(* CODESYS project Motor_4.2.6.0.library
   Company: ESO
   Description: Local Device Control - LDC Motor Library based on State Machine
   Version: 4.2.6.0
   Placeholder: ESO LDC Motor Library
   Author: Dan Popovic
   Title: ESO LDC Motor Library

Project tree, tasks and I/O mapping:
  libraries: ESO LDC Common Library, * (ESO); ESO LDC Timer Library, * (ESO); ESO MUDPI Library, * (ESO); Tc2_EtherCAT, * (Beckhoff Automation GmbH); Tc2_IoFunctions, * (Beckhoff Automation GmbH); Tc2_Math, * (Beckhoff Automation GmbH); Tc2_MC2, * (Beckhoff Automation GmbH); Tc2_MC2_Drive, * (Beckhoff Automation GmbH); Tc2_NC, * (Beckhoff Automation GmbH); Tc2_Standard, * (Beckhoff Automation GmbH); Tc2_System, * (Beckhoff Automation GmbH); Tc2_Utilities, * (Beckhoff Automation GmbH); Tc3_EventLogger, * (Beckhoff Automation GmbH); Tc3_Module, * (Beckhoff Automation GmbH); VisuDialogs, * (System); VisuSymbols, 3.5.10.0 (System)
  config/
    Mapping_with_new_EL6688_09_05.xml
    Mapping_with_old_EL6688_03_03.xml
    Mappings_SIM.xml
  00000000-0000-0000-0000-000000000000|config\Mapping_with_new_EL6688_09_05.xml
  00000000-0000-0000-0000-000000000000|config\Mapping_with_old_EL6688_03_03.xml
  00000000-0000-0000-0000-000000000000|config\Mappings_SIM.xml
  doc/
    AM8121_0F20_0000.xti
    EL7041_Phytron_57_500_1.2.xti
    EL7201_9014___AM8121_0F20_0000.xti
    MotorStateMachine.jpg
    Phytron_57_500_1.2_PID.xti
  00000000-0000-0000-0000-000000000000|doc\AM8121_0F20_0000.xti
  00000000-0000-0000-0000-000000000000|doc\EL7041_Phytron_57_500_1.2.xti
  00000000-0000-0000-0000-000000000000|doc\EL7201_9014___AM8121_0F20_0000.xti
  00000000-0000-0000-0000-000000000000|doc\MotorStateMachine.jpg
  00000000-0000-0000-0000-000000000000|doc\Phytron_57_500_1.2_PID.xti
  DUTs/
    Enumerated/
      Common/
        data type E_TIME_MODE
      Motor/
        data type E_DIRECTION
        data type E_MOTOR_AXIS_TYPE
        data type E_MOTOR_COMMAND
        data type E_MOTOR_ERROR
        data type E_MOTOR_EVENT
        data type E_MOTOR_INIT_ACTION
        data type E_MOTOR_INIT_SEQ_STATE
        data type E_MOTOR_INIT_STATE
        data type E_MOTOR_MODE
        data type E_MOTOR_MOVE_TYPE
        data type E_MOTOR_MOVING_STATE
        data type E_MOTOR_POST_INIT_STATE
        data type E_MOTOR_PRE_INIT_STATE
        data type E_MOTOR_RESET_STATE
        data type E_MOTOR_RPC_ERROR
        data type E_MOTOR_STATE
        data type E_MOTOR_STATUS
        data type E_MOTOR_SUBSTATE
        data type E_MOTOR_SWITCH_INDEX
      MultiAxis/
        data type E_MA_ADC_MOUNTING
        data type E_MA_AXES_ID
        data type E_MA_COMMAND
        data type E_MA_EVENT
        data type E_MA_MODE
        data type E_MA_ROTATOR_TYPE
        data type E_MA_RPC_ERROR
        data type E_MA_STATE
        data type E_MA_SUBSTATE
      Tracking/
        data type E_ADC_AXES_ID
        data type E_ADC_MODE
        data type E_DROT_MODE
        data type E_TRK_COMMAND
    Interfaces/
      interface ITrackCtrl: ComputeNextPos, HandleStates, Init, IsError, MoveInPos, MoveInSpeed, Reset
    Structures/
      Astro/
        data type E_ASTRO_TELESCOPE
        data type T_ASTRO_CCS_DATA
        data type T_ASTRO_DATA
        data type T_ASTRO_EL6688_DATA
        data type T_ASTRO_ENVIRONMENT
        data type T_ASTRO_MEAN_COORDINATES
        data type T_ASTRO_POLAR_MOTION
        data type T_ASTRO_SITE_CONSTANTS
        data type T_ASTRO_TIME
        data type T_ASTRO_TRACKING_DATA
      CCS_Sim/
        data type T_CCS_CFG
        data type T_CCS_CTRL
        data type T_CCS_STAT
      Common/
        data type T_PTP_TIME
        data type T_TIMEVAL
        data type T_UTC_TIME
      Motor/
        data type T_MOTOR_ACTIVE_LOW
        data type T_MOTOR_AXIS_CFG
        data type T_MOTOR_CFG
        data type T_MOTOR_CTRL
        data type T_MOTOR_INFO
        data type T_MOTOR_INIT_STEP
        data type T_MOTOR_MC_PARAMETER
        data type T_MOTOR_MOTION
        data type T_MOTOR_SIGNAL
        data type T_MOTOR_SPEED
        data type T_MOTOR_STAT
        data type T_MOTOR_SWITCHES
        data type T_POSITION
      MultiAxis/
        data type T_MA_CFG
        data type T_MA_CTRL
        data type T_MA_SM_STAT
        data type T_MA_STAT
        data type T_MA_TOUT_CFG
      Simulation/
        data type T_SIM_MOTOR_CFG
        data type T_SIM_MOTOR_STAT
      Tracking/
        data type T_ADC_CFG
        data type T_ADC_CMD
        data type T_ADC_CTRL
        data type T_ADC_INFO
        data type T_ADC_STAT
        data type T_ADC_UNIT_CFG
        data type T_ASTRO_COORDINATES
        data type T_DROT_CFG
        data type T_DROT_CTRL
        data type T_DROT_INFO
        data type T_DROT_STAT
  GVLs/
    global variables GVL_TrkDefaultEnvironment
    global variables GVL_TrkSiteConstants
  lib/
  POUs/
    Astro/
      function block FB_ASTRO [ST]: M_AstroDataUpdate, M_Configure, M_GetDec_ddmmss, M_GetRa_hhmmss, M_OffsetRaDec_arcsec, M_SetRaDec_hdmmss, M_TrkUpdate
    Functions/
      function F_astroDms2rad [ST]
      function F_astroHms2rad [ST]
      function F_astroRad2Dms [ST]
      function F_astroRad2Hms [ST]
      function F_astroSplitHms [ST]
      function F_atan2 [ST]
      function F_DCTIME64_TO_ULINT [ST]
      function F_MOD [ST]
      function F_RAD2DMS_STRING [ST]
      function F_RAD2HMS_STRING [ST]
      function F_slaPa [ST]
      function F_timeGetAbsoluteDcTime [ST]
      function F_timeGetDcTime [ST]
      function F_timeGetUTC [ST]
      function F_timeUTCToJD [ST]
      function F_timeUTCToMJD [ST]
      function F_vltMod [ST]
      function F_vltSign [ST]
    Misc/
      function block FB_DIGITAL_SIGNAL_FILTER [ST]
    Motor/
      function block FB_MOTOR [ST]: ActionClearNOVRAM, ActionErrExecute, ActionInitAbort, ActionInitComplete, ActionInitExecute, ActionInitReject, ActionMoveExecute, ActionResetExecute, ActionSetPosition, ActionStopExecute, ActionUnexpExecute, ActivityClearingNOVRAM, ActivityInitAborting, ActivityInitializing, ActivityMoving, ActivitySettingPosition, ActivityStopping, CheckForEvents, Dummy_UserExample, M_Configure, M_GetActualPos, M_GetOptimisedDistance, M_GetOptimisedPosition, M_GetRpcErrorText, M_HandleEnabled, M_MotorBrakeControl, M_MotorInitLock, M_MotorInitSeq, M_MotorPostInit, M_MotorPreInit, M_MotorReset, M_NormalizePos, M_NOVRAM_Clear, M_NOVRAM_Load, M_NOVRAM_Save, M_SetError, M_SetRpcStatus, M_UpdateSwitches, RPC_Disable, RPC_Enable, RPC_Init, RPC_MoveAbs, RPC_MoveRel, RPC_MoveVel, RPC_Reset, RPC_SetDebug, RPC_SetLog, RPC_Stop, UserPostInit, UserPostMove, UserPreInit, UserPreMove
      function block FB_MOTOR_BASE [ST]: ActionClearNOVRAM, ActionEnableExecute, ActionErrExecute, ActionInitAbort, ActionInitComplete, ActionInitExecute, ActionInitReject, ActionMoveExecute, ActionResetExecute, ActionSetPosition, ActionStopExecute, ActionUnexpExecute, ActivityClearingNOVRAM, ActivityInitAborting, ActivityInitializing, ActivityMoving, ActivitySettingPosition, ActivityStopping, CheckForEvents, M_CheckDisableIfUnsafe, M_GetErrorText, M_GetLogicalState, M_GetTimeInSec, M_LogEventDebug, M_LogEventEnd, M_LogEventError, M_LogEventGeneral, M_LogEventMoveAbs, M_LogEventMoveRel, M_LogEventMoveVel, M_LogEventStart, M_ReportFirstError, M_SetStatus, M_SetStatusDescription, ProcessEvents, SetAction, SetEvent, SetState, SetStatus
      function block FB_SIM_MOTOR [ST]: GetLogicalState, RPC_ResetConfig, RPC_SetCouplerState, RPC_SetDelay_Brake, RPC_SetDelay_SwitchActive, RPC_SetDelay_SwitchFind, RPC_SetFailure_BrakeFeedback
    MultiAxis/
      function block FB_MA_ADC [ST]: M_LogCommand, RPC_Disable, RPC_Enable, RPC_Init, RPC_MoveAbs, RPC_MoveAngle, RPC_MoveRel, RPC_MoveVel, RPC_Reset, RPC_StartTrack, RPC_Stop, RPC_StopTrack, User_ComputeAutoPos, User_ComputeNextPos, User_Configure, User_GetParams, User_SetParams
      function block FB_MA_BASE [ST]: ActionDisableExecute, ActionEnableExecute, ActionInitExecute, ActionMoveAbsExecute, ActionMoveVelExecute, ActionResetExecute, ActionStopExecute, ActionTrackExecute, ActivityDisabling, ActivityEnabling, ActivityInitialising, ActivityMoving, ActivityPresetting, ActivityResetting, ActivityStopping, ActivityTracking, CheckForEvents, M_AxesIdle, M_AxesInitialised, M_CheckAxesState, M_CheckError, M_Configure, M_GetMaxPosError, M_GetRpcErrorText, M_HomeMotors, M_LogCommand, M_LogEventError, M_LogEventGeneral, M_NextMove, M_NextMoveAbs, M_RestartTimer, M_SetInit, M_SetMode, M_SetRpcStatus, M_SetStatus, ProcessEvents, RPC_Init, SetAction, SetEvent, SetState, User_ComputeNextPos, User_Configure, User_GetParams, User_SetParams
      function block FB_MA_DROT [ST]: M_LogCommand, RPC_Disable, RPC_Enable, RPC_Init, RPC_MoveAbs, RPC_MoveAngle, RPC_MoveRel, RPC_MoveVel, RPC_Reset, RPC_StartTrack, RPC_Stop, RPC_StopTrack, RPC_TrackOffset, User_ComputeNextPos, User_Configure, User_GetParams, User_SetParams
      function block FB_TRK_BASE [ST]: User_Configure, User_GetParams, User_SetParams
    program MAIN [ST]
  Version/
    global variables Global_Version
  VISUs/
    Astro/
      visualisation GUI_ASTRO_CCS_SIM
    Motor/
      visualisation GUI_Motor001_Cfg
      visualisation GUI_Motor001_Ctrl
      visualisation GUI_Motor002_Cfg
      visualisation GUI_Motor002_Ctrl
    Templates/
      visualisation GUI_TEMPLATE_ASTRO_CCS_SIM
      visualisation GUI_TEMPLATE_MA_ADC
      visualisation GUI_TEMPLATE_MA_DROT
      visualisation GUI_TEMPLATE_MOTOR_CONFIG
      visualisation GUI_TEMPLATE_MOTOR_CONTROL
    Tracking/
      visualisation GUI_ADC_Motor1
      visualisation GUI_ADC_Motor2
      visualisation GUI_DROT_Cfg
      visualisation GUI_DROT_Motor
      visualisation GUI_MA_ADC
      visualisation GUI_MA_DROT
      visualisation GUI_TIMER
  global variables GCL
  text list GlobalTextList
  global variables GPL
*)

// DUTs/Enumerated/Common/E_TIME_MODE
{attribute 'qualified_only'}
{attribute 'strict'}
TYPE E_TIME_MODE :
(
	LOCAL	:= 0,
	UTC		:= 1
);
END_TYPE

// DUTs/Enumerated/Motor/E_DIRECTION
{attribute 'qualified_only'}
{attribute 'strict'}
TYPE E_DIRECTION :
(
	NEGATIVE := 1,
	POSITIVE
);
END_TYPE

// DUTs/Enumerated/Motor/E_MOTOR_AXIS_TYPE
{attribute 'qualified_only'}
{attribute 'strict'}
TYPE E_MOTOR_AXIS_TYPE :
(
	LINEAR				:= 1,
	CIRCULAR,
	CIRCULAR_OPTIMISED
);
END_TYPE

// DUTs/Enumerated/Motor/E_MOTOR_COMMAND
{attribute 'qualified_only'}
{attribute 'strict'}
TYPE E_MOTOR_COMMAND :
(
	NONE	:= 0,
	
	// Commands corresponding to events - MUST match E_MOTOR_EVENT !!!
	RESET,
	INIT,
	STOP,
	ENABLE,
	DISABLE,
	MOTOR_MOVE,
	SET_POSITION,
	CLEAR_NOVRAM
);
END_TYPE

// DUTs/Enumerated/Motor/E_MOTOR_ERROR
{attribute 'qualified_only'}
// 'strict' cannot be used since we mix our own codes with TC codes
//{attribute 'strict'}
TYPE E_MOTOR_ERROR :
(
	OK					:= 0,
	HW_NOT_OP,			
	LOCAL,			
	INIT_ABORTED,		
	TIMEOUT_INIT,
	TIMEOUT_MOVE,
	TIMEOUT_RESET,
	TIMEOUT_SETPOS,
	TIMEOUT_USER_PREINIT,
	TIMEOUT_USER_POSTINIT,
	TIMEOUT_USER_PREMOVE,
	TIMEOUT_USER_POSTMOVE,
	SETPOS,
	STOP,
	
	ABORT,
	SW_LIMIT_LOWER,
	SW_LIMIT_UPPER,
	BRAKE_ACTIVE,
	BRAKE_ENGAGE,
	BRAKE_DISENGAGE,
	SWITCH_NOT_USED,
	ENABLE,
	NOVRAM_READ,
	NOVRAM_WRITE,
	SWITCH_EXIT,
	STOP_LIMITS_BOTH,
	HW_LIMITS_BOTH,
	IN_POS,
	LOCKED,
	SoE_ADS_ERROR,
	SoE_SERCOS_ERROR,
	
	UNSAFE,		// EICSSW-1923

	// Simulator errors
	SIM_NOT_INITIALISED			:= 90,
	SIM_NULL_POINTER			:= 100,	

	// TwinCAT errors
	TC_VEL						:= 16929,	
	TC_NOT_READY_FOR_START		:= 16933,	
	TC_DISABLED_MOVE			:= 16992,	
	TC_BISECTION				:= 17022,	
	TC_MODULO_POS				:= 17026,	
	TC_STOP_ACTIVE				:= 17135,	
	TC_VEL_NEG					:= 17241,	
	TC_TARGET_LSW				:= 17504,	
	TC_TARGET_USW				:= 17505,	
	TC_FOLLOWING_ERROR			:= 17744,	
	TC_NOT_READY				:= 18000,	
	TC_IN_POS_6_SEC				:= 19207	

);
END_TYPE

// DUTs/Enumerated/Motor/E_MOTOR_EVENT
{attribute 'qualified_only'}
{attribute 'strict'}
TYPE E_MOTOR_EVENT :
(
	NONE	:= 0,
	
	(* events corresponding to commands - MUST match E_MOTOR_COMMAND *)
	RESET,
	INIT,
	STOP,
	ENABLE,
	DISABLE,
	MOTOR_MOVE,
	SET_POSITION,
	CLEAR_NOVRAM,
	
	(* 
		Events corresponding to internal events 
	*)
	
	MOVEDONE,		// Needed for detection of HW failures during initialisation
	STOPDONE,
	ENABLEDONE,
	DISABLEDONE,
	INITDONE,
	SETPOSDONE,
	

	HWOK,
	ERRLOCAL,
	ERRHW,
	ERRRESET,
	ERRFAULT,
	ERRINIT,
	ERRSTOP,
	ERRENABLE,
	ERRDISABLE,
	ERRBRAKE,
	ERRINPOS,
	ERRLOCKED,
	ERRTARGETPAR,
	ERRUSERPREINIT,
	ERRUSERPREMOVE,
	ERRUSERPOSTINIT,
	ERRUSERPOSTMOVE,
	TIMEOUT_MOVE,
	TIMEOUT_SETPOS,
	SW_LIMIT_LOWER,
	SW_LIMIT_UPPER,
	
	UNSAFE		// EICSSW-1923
	
);
END_TYPE

// DUTs/Enumerated/Motor/E_MOTOR_INIT_ACTION
TYPE E_MOTOR_INIT_ACTION :
(
	MOTOR_INIT_ACTION_END				:= 0,
	MOTOR_INIT_ACTION_FIND_INDEX,
	MOTOR_INIT_ACTION_FIND_REF_LE,
	MOTOR_INIT_ACTION_FIND_REF_UE,
	MOTOR_INIT_ACTION_FIND_LHW,
	MOTOR_INIT_ACTION_FIND_UHW,
	MOTOR_INIT_ACTION_DELAY,
	MOTOR_INIT_ACTION_MOVE_ABS,
	MOTOR_INIT_ACTION_MOVE_REL,
	MOTOR_INIT_ACTION_CALIB_ABS,
	MOTOR_INIT_ACTION_CALIB_REL,
	MOTOR_INIT_ACTION_CALIB_SWITCH,
	// The following steps cannot be configured in the INIT sequence
	MOTOR_INIT_ACTION_STEP1_START,
	MOTOR_INIT_ACTION_STEP1_EXECUTE,
	MOTOR_INIT_ACTION_STEP2_START,
	MOTOR_INIT_ACTION_STEP2_EXECUTE,
	MOTOR_INIT_ACTION_STOP
);
END_TYPE

// DUTs/Enumerated/Motor/E_MOTOR_INIT_SEQ_STATE
TYPE E_MOTOR_INIT_SEQ_STATE :
(
	MOTOR_INIT_SEQ_STATE_START				:= 0,
	MOTOR_INIT_SEQ_STATE_EXECUTE,
	MOTOR_INIT_SEQ_STATE_END
);
END_TYPE

// DUTs/Enumerated/Motor/E_MOTOR_INIT_STATE
TYPE E_MOTOR_INIT_STATE :
(
	MOTOR_INIT_STATE_START				:= 0,
	MOTOR_INIT_STATE_RESET,
	MOTOR_INIT_STATE_WAIT_READY,
	MOTOR_INIT_STATE_PRE_INIT,
	MOTOR_INIT_STATE_USER_PRE_INIT,
	MOTOR_INIT_STATE_INIT_SEQ,
	MOTOR_INIT_STATE_INIT_LOCK,
	MOTOR_INIT_STATE_POST_INIT,
	MOTOR_INIT_STATE_USER_POST_INIT,
	MOTOR_INIT_STATE_WAIT_BRAKE,
	MOTOR_INIT_STATE_SAVE_NOVRAM,
	MOTOR_INIT_STATE_END
);
END_TYPE

// DUTs/Enumerated/Motor/E_MOTOR_MODE
{attribute 'qualified_only'}
{attribute 'strict'}
TYPE E_MOTOR_MODE :
(
	POS				:= 0,
	VEL
);
END_TYPE

// DUTs/Enumerated/Motor/E_MOTOR_MOVE_TYPE
{attribute 'qualified_only'}
{attribute 'strict'}
TYPE E_MOTOR_MOVE_TYPE :
(
	NONE	:= 0,
	
	ABSOLUTE,
	RELATIVE,
	VELOCITY,
	TRACKING

);
END_TYPE

// DUTs/Enumerated/Motor/E_MOTOR_MOVING_STATE
TYPE E_MOTOR_MOVING_STATE :
(
	MOTOR_MOVING_STATE_NONE	:= 0,
	MOTOR_MOVING_STATE_ENABLE,
	MOTOR_MOVING_STATE_WAIT_BRAKES,
	MOTOR_MOVING_STATE_USER_PRE_MOVE,
	MOTOR_MOVING_STATE_WAIT_ABSOLUTE,
	MOTOR_MOVING_STATE_WAIT_OPTIMISED,
	MOTOR_MOVING_STATE_WAIT_VELOCITY,
	MOTOR_MOVING_STATE_USER_POST_MOVE,
	MOTOR_MOVING_STATE_APPLY_BRAKES,
	MOTOR_MOVING_STATE_DISABLE,
	MOTOR_MOVING_STATE_CHECK_IN_POS,
	MOTOR_MOVING_STATE_END
);
END_TYPE

// DUTs/Enumerated/Motor/E_MOTOR_POST_INIT_STATE
TYPE E_MOTOR_POST_INIT_STATE :
(
	MOTOR_POST_INIT_STATE_START	:= 0,
	MOTOR_POST_INIT_STATE_WRITE,
	MOTOR_POST_INIT_STATE_END
);
END_TYPE

// DUTs/Enumerated/Motor/E_MOTOR_PRE_INIT_STATE
TYPE E_MOTOR_PRE_INIT_STATE :
(
	MOTOR_PRE_INIT_STATE_START	:= 0,
	MOTOR_PRE_INIT_STATE_READ,
	MOTOR_PRE_INIT_STATE_GET_USER_UNITS,
	MOTOR_PRE_INIT_STATE_WRITE,
	MOTOR_PRE_INIT_STATE_END
);
END_TYPE

// DUTs/Enumerated/Motor/E_MOTOR_RESET_STATE
TYPE E_MOTOR_RESET_STATE :
(
	MOTOR_RESET_STATE_START	:= 0,
	MOTOR_RESET_STATE_SoE_RESET,
	MOTOR_RESET_STATE_SoE_WAIT_RESET,
	MOTOR_RESET_STATE_RESET_AXIS,
	MOTOR_RESET_STATE_WAIT,
	MOTOR_RESET_STATE_END
);
END_TYPE

// DUTs/Enumerated/Motor/E_MOTOR_RPC_ERROR
{attribute 'qualified_only'}
{attribute 'strict'}
TYPE E_MOTOR_RPC_ERROR :
(
	OK						:= 0,
	NOT_OP					:= -1,			
	NOT_NOTOP_READY			:= -2,			
	NOT_NOTOP_NOTREADY		:= -3,			
	LOCAL					:= -4,			
	SW_LIMIT_LOWER			:= -5,			
	SW_LIMIT_UPPER			:= -6,			
	INIT_WHILE_MOVING		:= -7,
	VEL_ZERO				:= -8,			
	VEL_NEG					:= -9,			
	VEL_MAX					:= -10,

	UNSAFE					:= -11	// EICSSW-1923			
);
END_TYPE

// DUTs/Enumerated/Motor/E_MOTOR_STATE
{attribute 'qualified_only'}
{attribute 'strict'}
TYPE E_MOTOR_STATE :
(
	NONE	:= 0,
	NOTOP,
	OP
);
END_TYPE

// DUTs/Enumerated/Motor/E_MOTOR_STATUS
{attribute 'qualified_only'}
{attribute 'strict'}
TYPE E_MOTOR_STATUS :
(
	OK	:= 0,
	ERROR,
	
	STANDING,
	MOVING

);
END_TYPE

// DUTs/Enumerated/Motor/E_MOTOR_SUBSTATE
{attribute 'qualified_only'}
{attribute 'strict'}
TYPE E_MOTOR_SUBSTATE :
(
	NONE					:= 0,
	
	NOTOP_NOTREADY			:= 100,
	NOTOP_READY				:= 101,
	NOTOP_INITIALIZING		:= 102,
	NOTOP_ABORTING			:= 107,
	NOTOP_CLEARING_NOVRAM	:= 108,
	
	NOTOP_ERROR				:= 199,
	
	
	OP_STANDSTILL			:= 216,            
	OP_MOVING				:= 217,
	OP_SETTING_POS			:= 218,
	OP_STOPPING				:= 219,
	
	OP_ERROR				:= 299
);
END_TYPE

// DUTs/Enumerated/Motor/E_MOTOR_SWITCH_INDEX
{attribute 'qualified_only'}
{attribute 'strict'}
TYPE E_MOTOR_SWITCH_INDEX :
(
	LSTOP	:= 0,
	LHW		:= 1,
	REF		:= 2,
	INDEX	:= 3,
	UHW		:= 4,
	USTOP	:= 5
);
END_TYPE

// DUTs/Enumerated/MultiAxis/E_MA_ADC_MOUNTING
TYPE E_MA_ADC_MOUNTING :
(
	// ADC positions should be the same due to oposite mounting of ADC units,
	// i.e. ADC2 = ADC1
	MA_ADC_MOUNTING_OPOSITE_SIDE := 0,
	// ADC positions should have oposite vales due to the same mounting of both ADC units,
	// i.e. ADC2 = -ADC1
	MA_ADC_MOUNTING_SAME_SIDE := 1
);
END_TYPE

// DUTs/Enumerated/MultiAxis/E_MA_AXES_ID
{attribute 'qualified_only'}
{attribute 'strict'}
TYPE E_MA_AXES_ID :
(
	ALL_AXES := 0,
	AXIS_1,
	AXIS_2,
	AXIS_3,
	AXIS_4,
	AXIS_5,
	AXIS_6
);
END_TYPE

// DUTs/Enumerated/MultiAxis/E_MA_COMMAND
{attribute 'qualified_only'}
{attribute 'strict'}
TYPE E_MA_COMMAND :
(
	NONE	:= 0,
	
	// Commands corresponding to events - MUST match E_MA_EVENT !!!
	RESET,
	INIT,
	STOP,
	ENABLE,
	DISABLE,
	MA_MOVE,
	START_TRACK,
	STOP_TRACK
);
END_TYPE

// DUTs/Enumerated/MultiAxis/E_MA_EVENT
{attribute 'qualified_only'}
{attribute 'strict'}
TYPE E_MA_EVENT :
(
	NONE	:= 0,
	
	(* events corresponding to commands - MUST match E_MA_COMMAND *)
	RESET,
	INIT,
	STOP,
	ENABLE,
	DISABLE,
	MA_MOVE,
	START_TRACK,
	STOP_TRACK,
	
	(* 
		Events corresponding to internal events 
	*)
	
	MOVEDONE,		// Needed for detection of HW failures during initialisation
	STOPDONE,
	ENABLEDONE,
	DISABLEDONE,
	INITDONE,
	TRACKDONE,
	TRACKEXIT,		// EICSSW-706: Tracking error >=  cfg.lrTrkThreshold => PRESETTING
	PRESETDONE,		// EICSSW-706: Presetting error < cfg.lrTrkThreshold => TRACKING
	

	HWOK,
	ERRLOCAL,
	ERRHW,
	
	UNSAFE		// EICSSW-1923
	
);
END_TYPE

// DUTs/Enumerated/MultiAxis/E_MA_MODE
TYPE E_MA_MODE :
(
	// WARNING: modes shall be a positive number
	MA_MODE_ENG	:= 0
);
END_TYPE

// DUTs/Enumerated/MultiAxis/E_MA_ROTATOR_TYPE
{attribute 'qualified_only'}
{attribute 'strict'}
TYPE E_MA_ROTATOR_TYPE :
(
	DROT 	:= 0,	// Derotator
	ADAPTER := 1,	// Adapter
	ROTATOR := 2	// Rotator
);
END_TYPE

// DUTs/Enumerated/MultiAxis/E_MA_RPC_ERROR
{attribute 'qualified_only'}
{attribute 'strict'}
TYPE E_MA_RPC_ERROR :
(
	OK						:=  0,
	NOT_OP					:= -1,			
	NOT_NOTOP_READY	    	:= -2,			
	NOT_NOTOP_NOTREADY		:= -3,			
	LOCAL					:= -4,			
	SW_LIMIT_LOWER			:= -5,			
	SW_LIMIT_UPPER			:= -6,			
	INIT_WHILE_MOVING		:= -7,
	VEL_ZERO				:= -8,			
	VEL_NEG					:= -9,			
	VEL_MAX					:= -10,
	NOT_TRACKING            := -11,

	UNSAFE					:= -12	// EICSSW-1923			
		
);
END_TYPE

// DUTs/Enumerated/MultiAxis/E_MA_STATE
{attribute 'qualified_only'}
//{attribute 'strict'}
TYPE E_MA_STATE :
(
	NONE	:= 0,
	NOTOP,
	OP
);
END_TYPE

// DUTs/Enumerated/MultiAxis/E_MA_SUBSTATE
{attribute 'qualified_only'}
//{attribute 'strict'}
TYPE E_MA_SUBSTATE :
(
	NONE				:=   0,
	
	NOTOP_NOTREADY		:= 100,
	NOTOP_READY			:= 101,
	NOTOP_INITIALISING	:= 102,
	NOTOP_ABORTING		:= 107,
	
	NOTOP_RESETTING		:= 109,
	NOTOP_ENABLING		:= 110,

	NOTOP_ERROR			:= 199,

	
	OP_DISABLING 		:= 205,
	OP_STANDSTILL		:= 216,            
	OP_MOVING			:= 217,
	OP_SETTING_POS		:= 218,
	OP_STOPPING			:= 219,
	OP_TRACKING			:= 220,
	OP_PRESETTING		:= 221,

	OP_ERROR			:= 299

);
END_TYPE

// DUTs/Enumerated/Tracking/E_ADC_AXES_ID
{attribute 'qualified_only'}
{attribute 'strict'}
TYPE E_ADC_AXES_ID :
(
	ALL_AXES := 0,
	ADC_1,
	ADC_2
);
END_TYPE

// DUTs/Enumerated/Tracking/E_ADC_MODE
{attribute 'qualified_only'}
{attribute 'strict'}
TYPE E_ADC_MODE :
(
	// WARNING: modes shall be a positive number
	ENG   := 0, 
	OFF   := 1,
	AUTO  := 2
);
END_TYPE

// DUTs/Enumerated/Tracking/E_DROT_MODE
{attribute 'qualified_only'}
{attribute 'strict'}
TYPE E_DROT_MODE :
(
	ENG		:= 0,
	STAT	:= 1,
	SKY		:= 2,
	ELEV	:= 3,
	USER	:= 4
);
END_TYPE

// DUTs/Enumerated/Tracking/E_TRK_COMMAND
{attribute 'qualified_only'}
{attribute 'strict'}
TYPE E_TRK_COMMAND :
(
	NONE			:= 0,
	INIT			:= 1,
	STOP, 
	TRK_MOVE,
	START_TRACK,
	STOP_TRACK,
	RESET,
	ENABLE,
	DISABLE,
	MOVE_MASTER
);
END_TYPE

// DUTs/Structures/Astro/E_ASTRO_TELESCOPE
{attribute 'qualified_only'}
{attribute 'strict'}
TYPE E_ASTRO_TELESCOPE :
(
	ELT := 0,
	UT1,
	UT2,
	UT3,
	UT4
);
END_TYPE

// DUTs/Structures/Astro/T_ASTRO_CCS_DATA
TYPE T_ASTRO_CCS_DATA :
STRUCT
	environment :	T_ASTRO_ENVIRONMENT;
	site :			T_ASTRO_SITE_CONSTANTS;
	motion :		T_ASTRO_POLAR_MOTION;
	dut :			LREAL;
	equinox :		LREAL;
	wavelength :	LREAL;
END_STRUCT
END_TYPE

// DUTs/Structures/Astro/T_ASTRO_DATA
TYPE T_ASTRO_DATA :
STRUCT
	time_data:			T_ASTRO_TIME;
	environment:		T_ASTRO_ENVIRONMENT;
	site:				T_ASTRO_SITE_CONSTANTS;
	motion:				T_ASTRO_POLAR_MOTION;
	mean:               T_ASTRO_MEAN_COORDINATES;
	tracking_data:		T_ASTRO_TRACKING_DATA;
	dut:             	LREAL := 0.0;
	equinox:			LREAL := 2000;
	wavelength:      	LREAL := 600;
END_STRUCT
END_TYPE

// DUTs/Structures/Astro/T_ASTRO_EL6688_DATA
TYPE T_ASTRO_EL6688_DATA :
STRUCT
	Control_value_update_toggle:	BOOL;
	External_device_not_connected:	BOOL;
	Internal_time_stamp:			ULINT;
	External_time_stamp:			ULINT;
END_STRUCT
END_TYPE

// DUTs/Structures/Astro/T_ASTRO_ENVIRONMENT
// Structure containing atmospheric conditions.
TYPE T_ASTRO_ENVIRONMENT :
STRUCT
	temperature:	LREAL   := 20.0;	// Air temperature [degC]
	pressure:		LREAL   := 760.0;	// Atmospheric Pressure [mbar]
	humidity:		LREAL   := 50;		// Relative humidity [0.0..1.0]
	lapserate:		LREAL   := 0.0065;
END_STRUCT
END_TYPE

// DUTs/Structures/Astro/T_ASTRO_MEAN_COORDINATES
TYPE T_ASTRO_MEAN_COORDINATES :
STRUCT
	alpha : 	LREAL := 0.0;
	delta : 	LREAL := -890000.0;
	epoch : 	LREAL;
	equinox : 	LREAL := 2000;
	pma : 		LREAL;
	pmd : 		LREAL;
	radvel : 	LREAL;
	parallax : 	LREAL;
END_STRUCT
END_TYPE

// DUTs/Structures/Astro/T_ASTRO_POLAR_MOTION
TYPE T_ASTRO_POLAR_MOTION :
STRUCT
	x : LREAL := 0.0;
	y : LREAL := 0.0;
END_STRUCT
END_TYPE

// DUTs/Structures/Astro/T_ASTRO_SITE_CONSTANTS
TYPE T_ASTRO_SITE_CONSTANTS :
STRUCT
	// Using Paranal Site configuration
	longitude :	LREAL := 1.228800386;
	latitude :	LREAL := -0.429833092;
	height :	LREAL := 2648;
END_STRUCT
END_TYPE

// DUTs/Structures/Astro/T_ASTRO_TIME
TYPE T_ASTRO_TIME :
STRUCT
	leap_second:	INT;
	lUtcTime:		ULINT;		   	// UTC time in nanoseconds
	sUtcTime:		STRING;			// UTC time as string
	ut1:			LREAL;			// MJD time [day]
	tu:				LREAL;			// TU  time [day]. tu := (ut1 - 51544.5) / 36525.0;
	gmst:			LREAL;			// Greenwich Mean Sidereal Time
	
END_STRUCT
END_TYPE

// DUTs/Structures/Astro/T_ASTRO_TRACKING_DATA
TYPE T_ASTRO_TRACKING_DATA :
STRUCT
	alt_r   : LREAL;	// altitude [rad]
	alt_deg : LREAL;	// altitude [deg]

	az_r    : LREAL;	// azimuth [rad]
	az_deg  : LREAL;	// azimuth [deg]

	ra_hms  : LREAL;	// RA  [Hms]
	ra_r    : LREAL;	// RA  [rad]
	ra_deg  : LREAL;	// RA  [deg]

	dec_dms : LREAL;	// Dec [Dms]
	dec_r   : LREAL;	// Dec [rad]
	dec_deg : LREAL;	// Dec [deg]

	pa_r    : LREAL;	// parallactic angle [rad]
	pa_deg  : LREAL;	// parallactic angle [deg]

	ha_hms  : LREAL;	// hour angle [Hms]
	ha_r    : LREAL;	// hour angle [rad]
	ha_deg  : LREAL;	// hour angle [deg]

	fr_r   	: LREAL;	// Field rotation [rad]
	fr_deg 	: LREAL;	// Field rotation [deg]
END_STRUCT
END_TYPE

// DUTs/Structures/CCS_Sim/T_CCS_CFG
TYPE T_CCS_CFG:
STRUCT
	site:     TrkSiteConstants;
END_STRUCT
END_TYPE

// DUTs/Structures/CCS_Sim/T_CCS_CTRL
TYPE T_CCS_CTRL:
STRUCT
	meanCoordinates: TrkMeanCoordinates;
	environment:     TrkEnvironment;
	motion:          TrkPolarMotion;
	wavelength:      LREAL := 600;
	dut:             LREAL := 0.0;
	equinox:         LREAL := 2000.0;
END_STRUCT
END_TYPE

// DUTs/Structures/CCS_Sim/T_CCS_STAT
TYPE T_CCS_STAT:
STRUCT
	apparent   :        TrkApparentCoordinates;
	observed   :        TrkObservedCoordinates;
	environment:        TrkEnvironment;
	data       :        TrkComputation;
	nTimeMode  :        DINT := 0;
	sTimeMode  :        STRING := '';
	sDcTime    :        STRING := '';
	lDcTime    :        LINT := 0;
END_STRUCT
END_TYPE

// DUTs/Structures/Common/T_PTP_TIME
(*
typedef struct _PTPTime
{
	ULONGLONG internal;
	ULONGLONG external;
	bool not_connected;
	bool update_toggle;
	LONGLONG dcTcOffset;
} PTPTime, *PPTPTime;
*)
TYPE T_PTP_TIME :
STRUCT
END_STRUCT
END_TYPE

// DUTs/Structures/Common/T_TIMEVAL
TYPE T_TIMEVAL :
STRUCT
    tv_sec:		UDINT;	// seconds since midnight January 1,1970 UTC
    tv_usec:	DINT;  	// and microseconds
END_STRUCT
END_TYPE

// DUTs/Structures/Common/T_UTC_TIME
TYPE T_UTC_TIME :
STRUCT
	dcTime:   ULINT;
	mode:     DINT;
END_STRUCT
END_TYPE

// DUTs/Structures/Motor/T_MOTOR_ACTIVE_LOW
TYPE T_MOTOR_ACTIVE_LOW :
STRUCT
	bValue:	BOOL	:= FALSE;
END_STRUCT
END_TYPE

// DUTs/Structures/Motor/T_MOTOR_AXIS_CFG
TYPE T_MOTOR_AXIS_CFG :
STRUCT
	////////////////////////////////////////////////////////////////////////
	// The following configuration parameters are read from Axis on INIT. //
	////////////////////////////////////////////////////////////////////////
	
	lrScaleFactor:	LREAL 	:= 1.0;				// Read from Axis on INIT
	lrModuloFactor: LREAL 	:= 360.0;			// Read from Axis on INIT
	lrAccel: 		LREAL 	:= 30.0;			// Read from Axis on INIT
	lrDecel: 		LREAL 	:= 30.0;			// Read from Axis on INIT
	lrJerk: 		LREAL 	:= 100;				// Read from Axis on INIT
	lrMaxVelocity:	LREAL 	:= 0.001;			// Read from Axis on INIT
	lrMaxPosLag:	LREAL 	:= 0.0;				// Read from Axis on INIT
	sUnits:			STRING(16) 	:= 'UNKNOWN';	// Read from Axis on INIT using ADS

END_STRUCT
END_TYPE

// DUTs/Structures/Motor/T_MOTOR_CFG
TYPE T_MOTOR_CFG :
STRUCT
	//////////////////////////////////////////////////////////
	// Parameters configurable from WS, Cfg GUI or directly //
	//////////////////////////////////////////////////////////
	
	// Backlash compensation value [UU], direction given by the sign, 
	// 0:	no backlash compensation, 
	// >0:	approach from positive direction, 
	// <0:	approach from negative direction
	lrBacklash:			LREAL 	:= 0.0;		
	lrDefaultVelocity:	LREAL 	:= 0.01;	// Default velocity for position mode [UU]

	// SW Limits.
	// If both limits are set to zero, limits are not used.
	lrMaxPosition:		LREAL 	:= 0.0;	//  [UU]
	lrMinPosition:		LREAL 	:= 0.0;	//  [UU]

	nAxisType:			DINT	:= E_MOTOR_AXIS_TYPE.LINEAR;

	// Timeouts
	nTimeoutInit:		UDINT 	:= 60000;	(* Timeout for complete INIT sequence [ms] *)
	nTimeoutMove:		UDINT 	:= 60000;	(* Timeout for a single move [ms] *)
	nTimeoutSwitch:		UDINT 	:= 15000;	(* Timeout for exiting a switch [ms] *)


	// Brake handling
	bUseBrake:			BOOL	:= FALSE;
	bActiveLowBrake:	BOOL	:= FALSE;

	// ActiveLow configuration for switches. Default is 'FALSE'. 
	bArrActiveLow:		ARRAY [E_MOTOR_SWITCH_INDEX.LSTOP..E_MOTOR_SWITCH_INDEX.USTOP] OF T_MOTOR_ACTIVE_LOW;
	
	// ActiveLow configuration for in-position switch. Default is 'FALSE'. 
	bActiveLowInPos:	BOOL	:= FALSE;

	// Default INIT sequence - Just calibrate to zero.
	strArrInitSeq:		ARRAY [1..10] OF T_MOTOR_INIT_STEP := [
											(nAction:=9, lrValue1:=0.0, lrValue2:=0.0),
											(nAction:=0, lrValue1:=0.0, lrValue2:=0.0),
											(nAction:=0, lrValue1:=0.0, lrValue2:=0.0),
											(nAction:=0, lrValue1:=0.0, lrValue2:=0.0),
											(nAction:=0, lrValue1:=0.0, lrValue2:=0.0),
											(nAction:=0, lrValue1:=0.0, lrValue2:=0.0),
											(nAction:=0, lrValue1:=0.0, lrValue2:=0.0),
											(nAction:=0, lrValue1:=0.0, lrValue2:=0.0),
											(nAction:=0, lrValue1:=0.0, lrValue2:=0.0),
											(nAction:=0, lrValue1:=0.0, lrValue2:=0.0)];
											
	// Function lock
	bLock:			BOOL	:= FALSE;	// If TRUE, motor is locked
	lrLockPos:		LREAL 	:= 0.0;		// Locked position [UU]
	lrLockTol:		LREAL 	:= 0.0;		// Tolerance for in-locked position [UU]
	
	// User defined methods execution
	bExecUserPreInit:	BOOL	:= FALSE;
	bExecUserPostInit:	BOOL	:= FALSE;
	bExecUserPreMove:	BOOL	:= FALSE;
	bExecUserPostMove:	BOOL	:= FALSE;
	
	// Misc checks
	bCheckInPos:		BOOL	:= FALSE;	// If TRUE, check if i_bInPos signal is active after move
	bDisableAfterMove:	BOOL	:= FALSE;	// If TRUE, disable motor after each move
	
	// SoE drives (Sercos over EtherCAT) , e.g. AX5000, need special Reset procedure FB_SoEReset()
	// in case of drive failure.
	// Other drives, i.e. CoE drives (Can over EtherCAT), are reset with the standard MC_Reset().
	// IMPORTANT NOTE: For the AX5000 the "Wait For WcState is OK" flag 
	//                 has to be activated in the Advanced EtherCAT Settings/General/Behavior.
	bSoE_Drive:			BOOL	:= FALSE;	// If TRUE, SoE drive, e.g. AX5000), default CoE, i.e. FALSE

	// Logging
	bLogExtTime:		BOOL 	:= FALSE;		// If TRUE, use external time in event logs. Default FALS
	bDebug:				BOOL 	:= FALSE;		// If TRUE, show event logs of Debug type. Default FALSE.
	bLog:				BOOL 	:= TRUE;		// If TRUE, log events. Default TRUE.
	
END_STRUCT
END_TYPE

// DUTs/Structures/Motor/T_MOTOR_CTRL
TYPE T_MOTOR_CTRL :
STRUCT
	// Command value and execution flag
	nCommand:	E_MOTOR_COMMAND	:= E_MOTOR_COMMAND.NONE;// See E_MOTOR_COMMAND 
	bExecute:	BOOL;									// Triggers command execution
	
	// If bLocalCmd is TRUE, commands are accepted in Local mode.
	// This var is set by each button press in local GUI.
	// This var is reset after each command handling.
	// Each button in local GUI has to have the first command:
	//    m_Instance.ctrl.bLocalCmd := TRUE;
	// This variable is not available in OPC UA namespace.
	//
	{attribute 'OPC.UA.DA' := '0'}
	bLocalCmd:		BOOL	:= FALSE;				

	// Motion parameters
	nMoveType:		DINT	:= E_MOTOR_MOVE_TYPE.NONE;
	nDirection:		DINT 	:= MC_Positive_Direction;
	lrPosition: 	LREAL 	:= 0.0;		// Value for MOVE_ABS
	lrOffset: 		LREAL 	:= 0.0;		// Value for MOVE_REL (EICSSW-781)
	lrVelocity:		LREAL 	:= 0.0001;

END_STRUCT
END_TYPE

// DUTs/Structures/Motor/T_MOTOR_INFO
TYPE T_MOTOR_INFO :
STRUCT
(*
Driver Information 

Change Log:
	0.1	2016-07-14	- Snapshot - Porting from FB_MOTOR_CONTROL.
		2016-07-14	- Snapshot - MC_Halt instead of MC_Stop.
					- Implemented NOVRAM Load/Save - to be tested.
					- Signals monitored during STOPPING in INIT.
					- Removed most of Lamp code (this was the starting point)
		2016-08-09	- Implemented NOVRAM R/W.
					- Both limit switches check done only after NOVRAM is loaded.
					- Created first Motor.library.
	0.2 2017-01-30	- Simulator FB_SIM_MOTOR improvements ONLY.
					- Addition of simulator status structure.
					- Improved recognition of INIT command.
					- Fixed handling of REF_LE signal level.
					- Addition of RPC calls.
	0.3 2017-06-23	- WARNING: Compatible with TC 3.1.4020 or later.
					- Addition of Simulator handling of STOP signals.
					- Additional checks for Move Done, i.e. CommandAborted and NotMoving.
					- Addition of method M_GetActualPos().
					- Normalise set position for circular-optimised.
					- Additional checks for STOP switches.
	0.4 2017-08-11	- Improved stopping using fbHalt().
					- STOP timeout increased from 3 to 10 sec.
					- Handling of E_MOTOR_EVENT.ERRSTOP while Stopping.
					- Direction disabled depending on L/U STOP active level - no relaxed case for INIT.
					- Addition of State Machine GUI.
	0.5 2017-08-31	- Big cleanup.
					- Removed unused cfg variables lrTolerance and lrToleranceEnc.
					- Removed unused cfg variable cfg.lrScaleFactor.
					- Renamed cfg.nTypeAxis to cfg.nAxisType.
					- Corrected stopping while searching for switches.
					- Renamed bActiveLow to bValue in T_MOTOR_ACTIVE_LOW. 
					- Removed stat.lrInPosTolerance.
					- Renamed stat.bLimSwitch* to stat.bStopSwitch*.
					- Removed E_MOTOR_HW_STATUS.
	0.6 2017-09-01	- Motor stopped on timeout in Position mode.
					- Removed substate E_MOTOR_SUBSTATE.OP_DISABLING.
	0.7 2017-09-07	- Completed RPC Calls.
	0.8 2017-10-06	- Addition of ctrl.bLocalCmd.
					- Addition of m_Instance.ctrl.bLocalCmd := TRUE; to each GUI button.
					- Addition of stat.nCounter 'alive' counter.
					- Addition of E_MOTOR_EVENT.ERRLOCAL.
					- Added check for stat.bLocal in RPC Calls.
					- Removed RPC_SetPos.
	0.9 2017-10-12	- Replaced nInternalEvent to nEvent in Activities.
					- Implemented handling of hitting SW limits.
					- Improved failure handling during INIT.
	0.10 2018-01-24	- Handling of Locked mode.
					- Addition of 'i_bInPos	AT %I*:	BOOL' signal for in-position check
					- Addition of config parameters for User Methods.
					- Addition of UserPreInit() and UserPostInit() methods.
					- Addition of UserPreMove() and UserPostMove() methods.
					- Added calls to UserPreInit() and UserPostInit() methods in ActivityInitializing().
					- Added calls to UserPreMove() and UserPostMove() methods in ActivityMoving().
					- Additonal configuration parameters in Config GUI.
					- Changed nCmdCycleCounter type from DINT to UDINT.
					- Implemented FB_MOTOR::M_NOVRAM_Clear().
					- Corrected handling of E_MOTOR_EVENT.STOP in E_MOTOR_SUBSTATE.NOTOP_*.
					- Implemented Auto Disable.
					- Implemented In-Position check
	0.11 2018-01-25	- Completed handling of Locked mode.
	0.12 2018-01-30	- If configured for Disable After Move, axis disabled after INIT.
					- Additions of ENABLE/DISABLE AXIS buttons.
	0.13 2018-02-02	- Addition of MOTOR_INIT_STATE_WAIT_READY state to wait for AxisReady after Reset.
	1.3.0.0			- Moved nCmdCycleCounter to T_MOTOR_STAT.
					- Addition of {attribute 'OPC.UA.DA' := '0'} to block unwanted FB's and vars.
					- Addition of {attribute 'OPC.UA.DA' := '0'} for all VAR_INST.
	1.4.0.0			- RPC calls return INT.
					- Addition of E_MOTOR_RPC_ERROR.
	1.5.0.0			- Renaming of methods - prefix M_.
					- Addition of M_GetErrorText() and M_SetStatusDescription().
					- Axis User Units read with ADSREAD.
					- Improved State Machine.
					- Addition of sLibVersion.
	1.7.0.0			- Check for SW Limits in RPC_MoveAbs() and RPC_MoveRel().
	1.8.0.0			- Added support for SoE Drives Reset.
	1.8.0.1			- Added stat.nCycleTime.
					- Added one cycle time to UTC coming from ASTRO.
	2.0.0.0			- Code grouped in subdirectories.
	2.1.0.0			- If not OP, motor goes to NOTOP_FAILURE.
					- Corrected simulator handling of CouplerStatus.
	2.2.0.0			- axisCfg structure moved to stat.axis.
					- Addition of stat.axis.lrMaxPosLag.
					- In case of both STOP or HW limits being active, motor goes to NOTOP_ERROR.
	2.3.0.0			- Going back to TC3.1.4022.14 due to increased library size.
					- Renaming States STANDBY->NOTOP & FAILURE->ERROR.
	3.0.0.0			- WARNING: Requires TwinCAT 3.1 build 4022.20 or higher.
					- Projects need Tc3_EventLogger library included in References.
					- Addition of Methods for Event Logs.
					- Addition of methods RPC_SetLog() and RPC_SetDebug().
					- Addition of cfg.bLog flag for enable/disable of logging.
					- Fixed bug with backlash in Circular-Optimised.
	3.0.0.1			- Addition of Debug Logs in INIT sequence.
	3.0.1.0			- Introduction of new command E_MOTOR_MOVE_TYPE.TRACKING.
					- Logs are disabled while tracking.
					- GVL.C_CYCLE_IDLE set to 10 allowing a minimum of 5 NC-Task SAF cycles for each command.
					  It is assumed that PlcTask cycle time 1 ms and NC-Task SAF cycle time is 2 ms.
					- Idle command cycles are compared with FB_MA::RefCfg.nMinSkipCycles rather than GVL.C_CYCLE_IDLE.
					- Addition of FB_MA::CmdMotorMoveTrk() that sends E_MOTOR_MOVE_TYPE.TRACKING command in tracking.
					- FB_MA::User_HandleExternalCmds is the only place where RefStat.nSkippedCycles is incremented.
					- ENG and OFF buttons on FB_MA_ADC GUI send TRK_CMD_STOP_TRACK instead of TRK_CMD_MOVE.
	3.0.1.1			- Renamed TC_EVENTS.OpsEventClass to TC_EVENTS.MotorOpsEventClass.
					- The EventClas must have unique name.
					- Warning: Don't use ver. 3.0.1.0.
	3.0.2.0			- Compiled with TC3.1.4022.27.
					- Solved problem of 'growing' libraries by setting 
					  Property/Advanced/BuildAction to None for Motor.library and pdf files in dir config.
					- Corrected string display of seconds in F_RAD2DMS_STRING and F_RAD2HMS_STRING.
*)
	sDate:			STRING(16)	:= '2019-04-26';
	sDescription:	STRING(64) 	:= 'State Machine based Motor control';
	sName:			STRING(16)	:= 'FB_MOTOR';
	sPlatform:		STRING(16)	:= 'CoDeSys';
	sSynopsis:		STRING(64)	:= 'General purpose motor controller';
	nVersionMajor:	DINT		:= 4;
	nVersionMinor:	DINT		:= 1;

END_STRUCT
END_TYPE

// DUTs/Structures/Motor/T_MOTOR_INIT_STEP
TYPE T_MOTOR_INIT_STEP :
STRUCT
	nAction:	DINT; 	(* e.g. FIND_LHW *)
	lrValue1:	LREAL;	(* Normally velocity *)
	lrValue2:	LREAL;	(* Normally position *)
END_STRUCT
END_TYPE

// DUTs/Structures/Motor/T_MOTOR_MC_PARAMETER
TYPE T_MOTOR_MC_PARAMETER :
STRUCT
	nNumber:	MC_AxisParameter;
	lrValue:	LREAL;
END_STRUCT
END_TYPE

// DUTs/Structures/Motor/T_MOTOR_MOTION
TYPE T_MOTOR_MOTION :
STRUCT
	motionType:	E_MOTOR_MODE;
	position:	T_POSITION;
	speed:		T_MOTOR_SPEED;
END_STRUCT
END_TYPE

// DUTs/Structures/Motor/T_MOTOR_SIGNAL
TYPE T_MOTOR_SIGNAL :
STRUCT
	bActive:	BOOL	:= FALSE;
	bActiveLow:	BOOL	:= FALSE;
	bUsed:		BOOL	:= FALSE;
	lrPosition:	LREAL	:= 0.0;
END_STRUCT
END_TYPE

// DUTs/Structures/Motor/T_MOTOR_SPEED
TYPE T_MOTOR_SPEED :
STRUCT
	value: 		LREAL;
	direction: 	MC_Direction;
END_STRUCT
END_TYPE

// DUTs/Structures/Motor/T_MOTOR_STAT
TYPE T_MOTOR_STAT :
STRUCT
	bLocal:			BOOL	:= FALSE;			// if TRUE, device operated from PLC GUI 
	nCounter:		UDINT	:= 0;				// Alive flag - increments on every PLC cycle
	nCmdCycleCounter:	UDINT := 0;				// Number of cycles since last command
	

	nLastCommand:	E_MOTOR_COMMAND		:= E_MOTOR_COMMAND.NONE;// Last command sent to the device 

	nErrorCode: 	E_MOTOR_ERROR 		:= E_MOTOR_ERROR.OK;	// Error code 
	nRpcErrorCode: 	E_MOTOR_RPC_ERROR 	:= E_MOTOR_RPC_ERROR.OK;// RPC Error code
	nStatus: 		E_MOTOR_STATUS		:= E_MOTOR_STATUS.OK;	// Device status 

	nState:			E_MOTOR_STATE		:= E_MOTOR_STATE.NOTOP;
	nSubstate:		E_MOTOR_SUBSTATE	:= E_MOTOR_SUBSTATE.NOTOP_NOTREADY;

	nMode:			E_MOTOR_MODE 		:= E_MOTOR_MODE.POS;	// Mode of operation, POS or VEL


	sErrorText: 	STRING 	:= 'OK'; 			// Error text 
	sRpcErrorText: 	STRING 	:= 'OK'; 			// RPC Error text 
	sStatus: 		STRING 	:= 'OK'; 			// Status in textual form, e.g. 'OFF' 
	sLibVersion:	STRING	:= 'UNKNOWN';		// Library version as string, e.g. '1.2.0.0'
	sFirstError:	string	:= '';				// First error to cause failure and to be logged
	
	sState:			STRING	:= 'NOT OP';
	sSubstate:		STRING	:= 'NOT READY';
	
	sActionDesc:	STRING	:= '';
	sEventDesc:		STRING	:= '';
	
	
	lrPosError:		LREAL := 0.0;	 	// Position error 
	lrPosTarget:	LREAL := 0.0;	 	// Target position adjusted to full Enc position 
	lrPosActual: 	LREAL;				// Actual position 
	lrScaleFactor:	LREAL;				// Scale [UU]/Enc
	lrVelActual: 	LREAL;				// Actual velocity 

	nBacklashStep:	DINT;	// Backlash step (1 or 2). If Backlash=0.0, motion starts from step 2.
	nInitStep:		DINT;	// Initialisation step in progress.
	nInitAction:	DINT;	// Passed to simulator to know if searching for limits
	
	// NOTE that the original Info Data is of type UINT, i.e. 16 bit unsigned.
	nInfoData1:		INT;	// Info Data 1 from Motor I/O terminal
	nInfoData2:		INT;	// Info Data 2 from Motor I/O terminal

	bAxisReady:		BOOL := FALSE;	// Flag if axis is ready
	bBrakeActive:	BOOL := FALSE;	// Flag if brake is active
	bEnabled:		BOOL := FALSE;	// Flag if axis is enabled
	bInitialised:	BOOL := FALSE;	// Flag if axis is initialised
	bInPosition:	BOOL := FALSE;	// Flag if axis is In-Position
	bStopSwitchPos:	BOOL := FALSE;	// Flag if LSTOP signal is active
	bStopSwitchNeg:	BOOL := FALSE;	// Flag if USTOP signal is active
	bLock:			BOOL := FALSE;	// Flag if motor is locked

	// Switch signals
	signals:		ARRAY [E_MOTOR_SWITCH_INDEX.LSTOP..E_MOTOR_SWITCH_INDEX.USTOP] OF T_MOTOR_SIGNAL;

	axis:			T_MOTOR_AXIS_CFG;	// Axis Config parameters - Read from TwinCAT Axis


END_STRUCT
END_TYPE

// DUTs/Structures/Motor/T_MOTOR_SWITCHES
TYPE T_MOTOR_SWITCHES :
STRUCT
(* Variables that need mapping *)
	bLSTOP:			BOOL;
	bLHW:			BOOL;
	bREF:			BOOL;
	bINDEX:			BOOL;
	bUHW:			BOOL;
	bUSTOP:			BOOL;
END_STRUCT
END_TYPE

// DUTs/Structures/Motor/T_POSITION
TYPE T_POSITION :
STRUCT
	number: LREAL;
END_STRUCT
END_TYPE

// DUTs/Structures/MultiAxis/T_MA_CFG
TYPE T_MA_CFG :
STRUCT
	nMinSkipCycles: DINT := GPL.C_CYCLE_IDLE;
	timeout:           T_MA_TOUT_CFG;
	lrTrkThreshold:	LREAL	:= 1.0;	// If maximum error is < this, bTrackingOK = TRUE
END_STRUCT
END_TYPE

// DUTs/Structures/MultiAxis/T_MA_CTRL
TYPE T_MA_CTRL :
STRUCT
	nCommand:		E_MA_COMMAND	:= E_MA_COMMAND.NONE; 
	bExecute:		BOOL;
	nMode:          INT;
END_STRUCT
END_TYPE

// DUTs/Structures/MultiAxis/T_MA_SM_STAT
TYPE T_MA_SM_STAT :
STRUCT
	sState:			STRING	:= 'NOT OP';
	sSubstate:		STRING	:= 'NOT READY';
	
	nState:			E_MA_STATE		:= E_MA_STATE.NOTOP;
	nSubstate:		E_MA_SUBSTATE	:= E_MA_SUBSTATE.NOTOP_NOTREADY;
	
	sActionDesc:	STRING	:= '';
	sEventDesc:		STRING	:= '';
END_STRUCT
END_TYPE

// DUTs/Structures/MultiAxis/T_MA_STAT
TYPE T_MA_STAT :
STRUCT
	bLocal:			    BOOL	:= FALSE;	    // if TRUE, device operated from PLC GUI 
	bInitialised:		BOOL    := FALSE;		// Flag if device is initialised
	bConfigured:		BOOL    := FALSE;		// Flag indicated that pointers to FB_MOTOR are set
	bTrackingOK:		BOOL	:= FALSE;		// if TRUE, Can switch from PRESETTING to TRACKING.
	bTrackingBAD:		BOOL	:= FALSE;		// if TRUE, Should switch from TRACKING back to PRESETTING. 

	nMode:		     	INT;
	sStatus:			STRING 	:= '';			(* Status description *)
	nStatus:            DINT    := 0;
	lrPosError:         LREAL;					// Highest difference (actualPos - targetPos)

	nErrorCode: 	    DINT    := E_MOTOR_ERROR.OK;	// Error code 
	nRpcErrorCode: 	    DINT 	:= E_MOTOR_RPC_ERROR.OK;			(* RPC Error code *)
	sRpcErrorText: 	    STRING 	:= 'OK'; 			// RPC Error text 
	
	sLibVersion:        STRING  := '';          (* Motor.library version *)

	sm:                  T_MA_SM_STAT;           // State machine status
	nCycleTime:			UDINT	:= 10000;		// Cycle time in [100ns], default 1 ms
	
	nSkippedCycles: 	DINT := 20;
END_STRUCT
END_TYPE

// DUTs/Structures/MultiAxis/T_MA_TOUT_CFG
// Configuration common to all axes in the Multi-Axis (MA) system.
// Configuration is gethered by comparing configuration of individual motors.
// These poarameters cannot be set from the WS.
TYPE T_MA_TOUT_CFG :
STRUCT
	nInitTimeout:     	UDINT := 60000;     // Default INIT timeout [ms]. The longest init time in the system.
	nMoveTimeout:     	UDINT := 60000;     // Default MOVE timeout [ms]. The longest init time in the system.
	nStopTimeout:     	UDINT := 10000;     // Default STOP timeout [ms]. The longest init time in the system.
END_STRUCT
END_TYPE

// DUTs/Structures/Simulation/T_SIM_MOTOR_CFG
TYPE T_SIM_MOTOR_CFG :
STRUCT
	bArrActiveLow:		ARRAY [E_MOTOR_SWITCH_INDEX.LSTOP..E_MOTOR_SWITCH_INDEX.USTOP] OF T_MOTOR_ACTIVE_LOW;
	bUseBrake:			BOOL	:= FALSE;
	bActiveLowBrake:	BOOL 	:= FALSE;
	
	// Action delays
	nDelay_SwitchFind:		UDINT := 5000;	// Delay for finding switch [ms]
	nDelay_SwitchActive:	UDINT := 3000;	// Delay for switch being active (exiting switch) [ms]
	nDelay_Brake:			UDINT :=  500;	// Delay for brake activation [ms]

	nCouplerState:			UINT := 8;		// HW state
END_STRUCT
END_TYPE

// DUTs/Structures/Simulation/T_SIM_MOTOR_STAT
TYPE T_SIM_MOTOR_STAT :
STRUCT
	bInitialised:	BOOL 	:= FALSE;
	nErrorCode: 	DINT 	:= E_MOTOR_ERROR.SIM_NOT_INITIALISED;	(* Error code *)
	sErrorText: 	STRING 	:= 'NOT INITIALISED'; 			(* Error text *)
	sStatus: 		STRING 	:= 'ERROR'; 					(* motor status in textual form, e.g. 'OK' or 'ERROR'*)
END_STRUCT
END_TYPE

// DUTs/Structures/Tracking/T_ADC_CFG
TYPE T_ADC_CFG EXTENDS T_MA_CFG :
STRUCT
	//
	// Configuration common to both ADC's.
	//
	lrPslope:       LREAL := 0.0023;		// Pressure slope [arcsec/mbar] (
	lrPoffset:		LREAL := 743.0;			// Default Pressure offset [mbar].
	lrTslope:       LREAL := -0.0061;		// Default Temperature slope [arcsec/degC]
	lrToffset:      LREAL := 12;			// Default Temperature offset [degC]
	lrAfactor:		LREAL := 3.32;			// ADC refraction factor [1/arcsec]
	lrZDlimit:      LREAL := 0.0174533;     // 1.0 deg Zenith Distance limit [rad]

	lrMinElev:      LREAL := 27.64;			// Minimum elevation [deg]


	// Specific configuration for each ADC unit, i.e. for each motor
	unitCfg:		ARRAY [1..2] OF T_ADC_UNIT_CFG;
END_STRUCT
END_TYPE

// DUTs/Structures/Tracking/T_ADC_CMD
TYPE T_ADC_CMD :
STRUCT
	motor_ctrl: T_MOTOR_CTRL;
END_STRUCT
END_TYPE

// DUTs/Structures/Tracking/T_ADC_CTRL
TYPE T_ADC_CTRL EXTENDS T_MA_CTRL :
STRUCT
	lrTargetPos:    ARRAY [1..2] OF LREAL;
	lrTargetVel:    LREAL;
	lrPosang: 		ARRAY [1..2] OF LREAL;
END_STRUCT
END_TYPE

// DUTs/Structures/Tracking/T_ADC_INFO
TYPE T_ADC_INFO :
STRUCT
	(* Driver Information *)
	sDate:			STRING(32)	:= '2017-07-19';
	sDescription:	STRING(80) 	:= 'ADC control';
	sName:			STRING(64)	:= 'FB_ADC';
	sPlatform:		STRING(32)	:= '';
	sSynopsis:		STRING(64)	:= '';
	nVersionMajor:	DINT		:= 0;
	nVersionMinor:	DINT		:= 1;
END_STRUCT
END_TYPE

// DUTs/Structures/Tracking/T_ADC_STAT
TYPE T_ADC_STAT EXTENDS T_MA_STAT :
STRUCT
	lrPos:			 	LREAL   := 0.0;
	lrAdaPosAngle:      LREAL   := 0.0;
	lrDrotPos:          LREAL   := 0.0;
	lrRa:               LREAL   := 0.0;
	lrDec:              LREAL   := 0.0;
	lrAlt:              LREAL   := 0.0;
	lrAz:               LREAL   := 0.0;
	lrPa:               LREAL   := 0.0;
END_STRUCT
END_TYPE

// DUTs/Structures/Tracking/T_ADC_UNIT_CFG
TYPE T_ADC_UNIT_CFG :
STRUCT
	nSignOff:   	DINT  := 1;				// sign, e.g. ADC position sign for OFF  mode
	nSignAuto:      DINT  := 1;				// sign, e.g. ADC position sign for AUTO mode
	nSignPhi: 	    DINT  := 1;				// sign, e.g. ADC sign for phi (refraction) component

	lrRefOff:       LREAL := 0.0;			// Reference (offset) for OFF  mode
	lrRefAuto:      LREAL := 0.0;			// Reference (offset) for AUTO mode

	lrCoffset:		LREAL := 1.7387;		// Default C offset [arcsec]
	lrPosOffset:    LREAL := 90;			// Default Position offset [deg]
	lrDrotFactor:   LREAL := 2;				// Derotator factor

END_STRUCT
END_TYPE

// DUTs/Structures/Tracking/T_ASTRO_COORDINATES
TYPE T_ASTRO_COORDINATES :
STRUCT
	alpha: LREAL := 0;		// [hms]
	delta: LREAL := 0;		// [dms]
END_STRUCT
END_TYPE

// DUTs/Structures/Tracking/T_DROT_CFG
TYPE T_DROT_CFG EXTENDS T_MA_CFG :
STRUCT
	nFocusSign: 	DINT  := -1;             (* Sign 2 in LCU code *)
	nDirSign:   	DINT  := 1;              (* Sign 1 in LCU code *)
	lrSkyRef:    	LREAL := 0;              (* SKY reference position  *)
    lrElevRef:   	LREAL := 0;              (* ELEV reference position *)
	lrStatRef:   	LREAL := 0;              (* STAt reference position *)
	lrUserRef:   	LREAL := 0;              (* USER reference position *)
	lrUserPar1:  	LREAL := 0;				 (* User parameter 1        *)
	lrUserPar2:  	LREAL := 0;				 (* User parameter 2        *)
	lrUserPar3:  	LREAL := 0;				 (* User parameter 3        *)
	lrUserPar4:     LREAL := 0;              (* User parameter 4        *)
END_STRUCT
END_TYPE

// DUTs/Structures/Tracking/T_DROT_CTRL
TYPE T_DROT_CTRL EXTENDS T_MA_CTRL :
STRUCT
	lrTargetPos:    LREAL;
	lrTargetVel:    LREAL;
	lrPosang: 		LREAL;
	lrUserPar1:     LREAL := 0.0;
	lrUserPar2:     LREAL := 0.0;
	lrUserPar3:     LREAL := 0.0;
	lrUserPar4:     LREAL := 0.0;
	lrRotation:     LREAL := 0.0;
	lrOffset:       LREAL := 0.0;
	lrPupil:        LREAL := 0.0;
	lrParallactic:  LREAL := 0.0;
END_STRUCT
END_TYPE

// DUTs/Structures/Tracking/T_DROT_INFO
TYPE T_DROT_INFO :
STRUCT
	(* Driver Information *)
	sDate:			STRING(32)	:= '2017-07-19';
	sDescription:	STRING(80) 	:= 'Drotator control';
	sName:			STRING(64)	:= 'FB_DROT';
	sPlatform:		STRING(32)	:= '';
	sSynopsis:		STRING(64)	:= '';
	nVersionMajor:	DINT		:= 0;
	nVersionMinor:	DINT		:= 1;
END_STRUCT
END_TYPE

// DUTs/Structures/Tracking/T_DROT_STAT
TYPE T_DROT_STAT EXTENDS T_MA_STAT :
STRUCT
	lrRotation:         LREAL   := 0;
	lrPupil:            LREAL   := 0;
	lrAngleOnSky:       LREAL   := 0;
	lrModeAngle:        LREAL   := 0;
	lrActualVel:        LREAL;
	lrPosAng:           LREAL   := 0.0;
	lrPos:			 	LREAL   := 0.0;
	lrTotalOffset:	    LREAL   := 0.0;
	lrUserPar1:         LREAL;
	lrUserPar2:         LREAL;
	lrUserPar3:         LREAL;
	lrUserPar4:         LREAL;
END_STRUCT
END_TYPE

// GVLs/GVL_TrkDefaultEnvironment
{attribute 'qualified_only'}
VAR_GLOBAL
	C_HUMIDITY:    LREAL := 50.0;
	C_LAPSERATE:   LREAL := 0.0065;
	C_PRESSURE:    LREAL := 760.0;
	C_TEMPERATURE: LREAL := 20;
END_VAR

// GVLs/GVL_TrkSiteConstants
{attribute 'qualified_only'}
VAR_GLOBAL
	C_HEIGHT    : LREAL := 2648;
	C_LONGITUDE : LREAL := 1.228800386;
	C_LATITUDE  : LREAL := -0.429833092;
END_VAR

// Version/Global_Version
{attribute 'TcGenerated'}
{attribute 'no-analysis'}
{attribute 'linkalways'}
// This function has been automatically generated from the project information.
VAR_GLOBAL CONSTANT
	{attribute 'const_non_replaced'}
	stLibVersion_ESO_LDC_Motor_Library : ST_LibVersion := (iMajor := 4, iMinor := 2, iBuild := 6, iRevision := 0, nFlags := 0, sVersion := '4.2.6.0');
END_VAR

// GCL
{attribute 'qualified_only'}
VAR_GLOBAL CONSTANT
    C_PI:				LREAL := 3.1415926535897932384626433832795028841971693993751;
    C_PI2: 				LREAL := C_PI / 2.0;
	C_2PI: 				LREAL := 2.0 * C_PI;
	C_RAD2DEG:  		LREAL := (180.0 / C_PI);
	C_DEG2RAD:  		LREAL := (C_PI / 180.0);
	// pi/(12*3600):  seconds OF TIME TO radians */
	C_S2R:				LREAL := 7.2722052166430399038487115353692196393452995355905E-5;

	C_DIAG_COE_IDX: 	WORD  := 16#FA80; 	// EL_6688 CoE address for diagnostic data
	C_UTC_OFFSET_SIDX: 	BYTE  := 11;		// EL_6688 CoE subindex for UTC offset - Leap second
	C_PTP_OFFSET_SIDX: 	BYTE  := 6;			// EL_6688 Coe subindex for PTP offset from master

	C_KELVIN:			LREAL := 273.15;	// Zero deg C expressed in [deg K]
	C_MAX_P:    		LREAL := 900.0;		// Maximum pressure [mbar]
	C_MIN_P:    		LREAL := 600.0;		// Minimum pressure [mbar]
	C_MAX_T:    		LREAL := 50.0;		// Maximum temperature [deg C]
	C_MIN_T:			LREAL := -20.0;		// Minimum temperature [deg C]
	
	C_LATITUDE_ELT:		LREAL := -0.429165991;	// ELT Latitude  [rad]
	C_LATITUDE_VLT_UT1:	LREAL := -0.429833092;	// VLT_UT1 Latitude [rad] -24 deg 37 min 39.44 sec
	C_LATITUDE_VLT_UT2:	LREAL := -0.429825122;	// VLT_UT2 Latitude [rad] -24 deg 37 min 37.80 sec
	C_LATITUDE_VLT_UT3:	LREAL := -0.429819523;	// VLT_UT3 Latitude [rad] -24 deg 37 min 36.64 sec
	C_LATITUDE_VLT_UT4:	LREAL := -0.429823005;	// VLT_UT4 Latitude [rad] -24 deg 37 min 37.36 sec
	C_LATITUDE_NTT:		LREAL := -0.5106547351;	// NTT Latitude  [rad]
	C_LATITUDE_VISTA:	LREAL := -0.4296250041;	// VISTA Latitude  [rad] -24 36 56.518226
	C_LATITUDE_VST:		LREAL := -0.429788783;	// VST Latitude  [rad] -24 deg 37 min 30.300 sec
	C_LATITUDE_VLT_CM:	LREAL := -0.429833092;	// VLT_CM Latitude  [rad]

	C_LONGITUDE_ELT:	LREAL :=  1.225074527;	// ELT Longitude [rad]
	C_LONGITUDE_VLT_UT1:LREAL :=  1.228800386;	// VLT_UT1 Longitude [rad] 70 deg 24 min 18.27 sec
	C_LONGITUDE_VLT_UT2:LREAL :=  1.228796107;	// VLT_UT2 Longitude [rad] 70 deg 24 min 17.39 sec
	C_LONGITUDE_VLT_UT3:LREAL :=  1.228790929;	// VLT_UT3 Longitude [rad] 70 deg 24 min 16.32 sec
	C_LONGITUDE_VLT_UT4:LREAL :=  1.228780856;	// VLT_UT4 Longitude [rad] 70 deg 24 min 14.25 sec
	C_LONGITUDE_NTT:	LREAL :=  1.2345499197;	// NTT Longitude [rad]
	C_LONGITUDE_VISTA:	LREAL :=  1.2286692091;	// VISTA Longitude [rad] 70 23 51.216354
	C_LONGITUDE_VST:	LREAL :=  1.228759771;	// VST Longitude [rad] 70 deg 24 min 09.896 sec
	C_LONGITUDE_VLT_CM:	LREAL :=  1.228800386;	// VLT_CM Longitude [rad]

	
	C_LEAP_SECOND:		DINT  := 37;		// Last known Leap Second
	
	C_OFFSET_UNIX:		DINT  :=  946684800;  // seconds between years 1970 and 2000 


	C_CONST1:		LREAL :=  1721013.5;      // CONSTANT used in formula
	C_CONST2:		LREAL :=  190002.5;       // CONSTANT used in formula
	C_CONST3:		LREAL :=  2400000.5;      // CONSTANT used in formula
	C_CONST4:		LREAL :=  2440587.5;      // JD FOR 1970-01-01 00:00:00.000000


//#define vltMOD(A,B) ((B)!=0.0?((A)*(B)>0.0?(A)-(B)*floor_((A)/(B)):(A)+(B)*floor_(-(A)/(B))):(A))


END_VAR

// GPL
{attribute 'qualified_only'}
VAR_GLOBAL CONSTANT
	C_CYCLE_IDLE: 		DINT  := 10;		// Minimum number of idle cycles between commands to motor

    C_POS_SPEED: 		LREAL := 3;			// TODO ?
    C_MAX_SPEED: 		LREAL := 5;			// TODO ?
	C_MIN_SPEED: 		LREAL := 0.01;		// TODO ?

	C_MA_MAX_AXES:		INT 	:= 6;			// Maximum number of axes
	
END_VAR

// DUTs/Interfaces/ITrackCtrl
INTERFACE ITrackCtrl

METHOD ComputeNextPos : BOOL
VAR_INPUT
END_VAR

VAR_OUTPUT
	newPos : LREAL;
END_VAR
END_METHOD

METHOD HandleStates : BOOL
VAR_INPUT
END_VAR
END_METHOD

METHOD Init : BOOL
VAR_INPUT
END_VAR
END_METHOD

METHOD IsError : BOOL
VAR_INPUT
END_VAR
END_METHOD

METHOD MoveInPos : BOOL
VAR_INPUT
	refMotion: REFERENCE TO T_MOTOR_MOTION;
END_VAR
END_METHOD

METHOD MoveInSpeed
VAR_INPUT
	refMotion: REFERENCE TO T_MOTOR_MOTION;
END_VAR
END_METHOD

METHOD Reset : BOOL
VAR_INPUT
END_VAR
END_METHOD

END_INTERFACE

// POUs/Astro/FB_ASTRO
FUNCTION_BLOCK FB_ASTRO
VAR_INPUT
	in_TimeStat:		REFERENCE TO T_TIME_STAT;	// REF to FB_TIMER.stat
	in_Ra_hhmmss:		LREAL	:= 0.0;
	in_Dec_ddmmss:		LREAL	:= -890000.0;
	in_nTel:			E_ASTRO_TELESCOPE	:= E_ASTRO_TELESCOPE.ELT;
END_VAR
VAR_OUTPUT
	// CCS Deterministic data that normally come 
	// from the Telescope via MUDPI interface.
	{attribute 'OPC.UA.DA' := '0'}
	out_CcsDeterministic:	T_ASTRO_POINTING_KERNEL_POSITIONS;
END_VAR
VAR

	// All data calculated in FB_ASTRO
	{attribute 'OPC.UA.DA' := '0'}
	AstroData: 				T_ASTRO_DATA;	
    UserPointingKernel: 	T_ASTRO_POINTING_KERNEL_POSITIONS;		
 
	
	{attribute 'OPC.UA.DA' := '0'}
	q_trk_data          AT %Q*: T_ASTRO_POINTING_KERNEL_POSITIONS;

	bConfigured:	BOOL;
	
END_VAR

// Copy input variables on start
M_Configure();

//
// Update all input parameters into AstroData structure.
//
M_AstroDataUpdate();

//
// Update tracking data, i.e. gmst, ra, dec, alt, az, pa, ha, etc.
// Update also CcsDeterministic output structure.
//
M_TrkUpdate();

// Set outputs for mapping.
q_trk_data	:= out_CcsDeterministic;

METHOD M_AstroDataUpdate
VAR_INPUT
END_VAR
END_METHOD

METHOD M_Configure
VAR_INPUT
END_VAR
IF NOT bConfigured	THEN
	bConfigured	:= TRUE;
	
	AstroData.mean.alpha	:= in_Ra_hhmmss;
	AstroData.mean.delta	:= in_Dec_ddmmss;
	
	// Set telescope coordinates
	CASE in_nTel OF 
		E_ASTRO_TELESCOPE.ELT:
			AstroData.site.longitude	:= F_astroDms2rad( 701119.20);
			AstroData.site.latitude		:= F_astroDms2rad(-243511.99);
			AstroData.site.height		:= 3046.0;
		
		E_ASTRO_TELESCOPE.UT1:
			AstroData.site.longitude	:= F_astroDms2rad( 702418.27);
			AstroData.site.latitude		:= F_astroDms2rad(-243739.44);
			AstroData.site.height		:= 2635.0;
		
		E_ASTRO_TELESCOPE.UT2:
			AstroData.site.longitude	:= F_astroDms2rad( 702417.39);
			AstroData.site.latitude		:= F_astroDms2rad(-243737.80);
			AstroData.site.height		:= 2635.0;
		
		E_ASTRO_TELESCOPE.UT3:
			AstroData.site.longitude	:= F_astroDms2rad( 702416.32);
			AstroData.site.latitude		:= F_astroDms2rad(-243736.64);
			AstroData.site.height		:= 2635.0;
		
		E_ASTRO_TELESCOPE.UT4:
			AstroData.site.longitude	:= F_astroDms2rad( 702414.24);
			AstroData.site.latitude		:= F_astroDms2rad(-243737.36);
			AstroData.site.height		:= 2635.0;
		
	END_CASE

END_IF
END_METHOD

METHOD M_GetDec_ddmmss : LREAL
VAR_INPUT
END_VAR
M_GetDec_ddmmss	:= AstroData.mean.delta;
END_METHOD

METHOD M_GetRa_hhmmss : LREAL
VAR_INPUT
END_VAR
M_GetRa_hhmmss	:= AstroData.mean.alpha;
END_METHOD

// Set Ra and Dec offsets in arcsec
METHOD M_OffsetRaDec_arcsec
VAR_INPUT
	in_lrOffsetRa_arcsec:	LREAL;	// Offset in Ra  [arcsec]
	in_lrOffsetDec_arcsec:	LREAL;	// Offset in Dec [arcsec]
END_VAR
VAR
	lrTmp:			LREAL;
	lrOffset_rad:	LREAL;	// Offset in [rad].
	lrOffset_h:		LREAL;	// Offset in [h].
END_VAR
//
// Ra offset
//

// Get Ra in rad
lrTmp	:= F_astroHms2rad(AstroData.mean.alpha);

// Convert arcsec->hour
lrOffset_h	:= in_lrOffsetRa_arcsec / 3600.0 * 24 / 360.0;

// Conversion h->rad
lrOffset_rad	:= lrOffset_h / 24.0 * 2*PI;

// Add the offset to the current Ra value in rad
lrTmp	:= lrTmp + lrOffset_rad;

// Convert rad to hhmmss.
AstroData.mean.alpha	:= F_astroRad2Hms(lrTmp);


//
// Dec offset
//

// Get Dec in rad
lrTmp	:= F_astroDms2rad(AstroData.mean.delta);

// Get the Dec offset in rad first.
// Conversion: arcsec->deg, and then deg->rad.
lrOffset_rad	:= (in_lrOffsetDec_arcsec / 3600.0) * PI / 180.0;

// Add the offset to the current Dec value in rad
lrTmp	:= lrTmp + lrOffset_rad;

// Convert rad to ddmmss.
AstroData.mean.delta	:= F_astroRad2Dms(lrTmp);
END_METHOD

// Set Ra in hhmmss.sss and Dec in ddmmss.sss
METHOD M_SetRaDec_hdmmss
VAR_INPUT
	in_lrRa:	LREAL;	// Ra  [hhmmss.sss]
	in_lrDec:	LREAL;	// Dec [ddmmss.sss]
END_VAR
AstroData.mean.alpha	:= in_lrRa;
AstroData.mean.delta	:= in_lrDec;
END_METHOD

METHOD M_TrkUpdate : BOOL
VAR_INPUT
END_VAR
VAR
	ra_r, dec_r:	LREAL;
	temp1, temp2, temp3, temp4:	LREAL;
	ut1, t, tu, A:	LREAL;
	
	sh, ch, cd, chcd, sp, sdcp, cp, sd, x, y, rsq:	LREAL;

	track:	REFERENCE TO T_ASTRO_TRACKING_DATA;
	coord:	REFERENCE TO T_ASTRO_SITE_CONSTANTS;
	time_data:	REFERENCE TO T_ASTRO_TIME;
	
	latitude, longitude:	LREAL;
	
END_VAR
// This is the slalib C code translated into ST.
//
// HRESULT TrkUpdate()
//

//
// Set references to output data structures
//
track		REF=AstroData.tracking_data;
coord		REF=AstroData.site;
time_data	REF=AstroData.time_data;


// Copy ra and dec from input to output data structures
track.ra_hms  := AstroData.mean.alpha;
track.dec_dms := AstroData.mean.delta;

// Get ra and dec in radians and degrees
track.ra_r		:= F_astroHms2rad(track.ra_hms);
track.ra_deg	:= track.ra_r * GCL.C_RAD2DEG;
track.dec_r		:= F_astroDms2rad(track.dec_dms);
track.dec_deg	:= track.dec_r * GCL.C_RAD2DEG;

ra_r	:= track.ra_r;
dec_r	:= track.dec_r;
	

latitude	:= AstroData.site.latitude;
longitude	:= AstroData.site.longitude;

temp1 := COS(dec_r) * TAN(latitude);
temp2 := SIN(dec_r);
temp3 := temp2 * SIN(latitude);
temp4 := COS(dec_r) * COS(latitude);


//
// Calculate times
//
ut1 := F_timeUTCToMJD(F_timeGetUTC(in_TimeStat.lUtcTime));	
tu := (ut1 - 51544.5) / 36525.0;

// Updata T_ASTRO_TIME structure
time_data.leap_second	:= in_TimeStat.el6688.diagnostics.leap_second;
IF time_data.leap_second = 0	THEN
	time_data.leap_second	:= 37;
END_IF
time_data.lUtcTime		:= in_TimeStat.lUtcTime;
time_data.sUtcTime		:= in_TimeStat.sUtcTime;
time_data.ut1			:= ut1;
time_data.tu			:= tu;

time_data.gmst :=	F_vltMOD(ut1, 1.0) * GCL.C_2PI +
				(24110.54841 + (8640184.812866 + (0.093104 - 6.2E-6 * tu) * tu) * tu) * GCL.C_S2R;
time_data.gmst := F_vltMOD(time_data.gmst, GCL.C_2PI);

IF time_data.gmst < 0.0 THEN
	time_data.gmst := time_data.gmst + GCL.C_2PI;
END_IF

//
// Hour angle
//
track.ha_r := time_data.gmst - (longitude + ra_r);	// TODO: Check the formula

// Hour angle is in range 0..2PI [rad], i.e. 0..24 [hour]
IF track.ha_r > GCL.C_2PI THEN
	track.ha_r	:= track.ha_r - GCL.C_2PI;
ELSIF track.ha_r < 0.0 THEN
	track.ha_r	:= track.ha_r + GCL.C_2PI;
END_IF

track.ha_deg	:= track.ha_r * GCL.C_RAD2DEG;
track.ha_hms	:= F_astroRad2Hms(track.ha_r);

//
// CALC. parallactic angle 
//
// t = tan(latitude) * cos(dec) - sin(dec) * cos(hourAngle); 
t := temp1 - temp2 * COS(track.ha_r);
IF t = 0.0 THEN
	M_TrkUpdate := FALSE;  // error 
	RETURN;
END_IF


// 
// Parallactic angle
// 
track.pa_r := F_slaPa(track.ha_r, dec_r, latitude);

// Original PA calculation
track.pa_r := ATAN(SIN(track.ha_r) / t) + GCL.C_PI;
track.pa_r := F_vltMod(GCL.C_PI2 * F_vltSign(t) + track.pa_r + GCL.C_PI2 , GCL.C_2PI) +
					GCL.C_PI2 * (-F_vltSign(track.ha_r) + 1) * 
				  (F_vltSign(dec_r - latitude) - 1);	
// Keep -PI < PA < PI
IF track.pa_r > GCL.C_PI THEN
	track.pa_r := track.pa_r - GCL.C_2PI;
ELSIF track.pa_r < -GCL.C_PI THEN
	track.pa_r := track.pa_r + GCL.C_2PI;
END_IF

track.pa_deg := track.pa_r * GCL.C_RAD2DEG;


//
// CALC. telescope altitude in radians and degrees.
//
// altitude = asin(sin(dec) * sin(latitude) + cos(dec) * cos(latitude) * cos(hourAngle));
track.alt_r := ASIN(temp3 + temp4 * COS(track.ha_r));
track.alt_deg := track.alt_r * GCL.C_RAD2DEG;

//
// DPO: slaE2h()
//
(*
	* A = acos((sin(dec) - sin(altitude) * sin(latitude))
	*             ---------------------------------------
	*			      cos(altitude)*cos(latitude))
*)
sh := SIN(track.ha_r);
ch := COS(track.ha_r);
sd := SIN(dec_r);
cd := COS(dec_r);
sp := SIN(latitude);
cp := COS(latitude);
chcd := ch * cd;
sdcp := sd * cp;
x := - chcd * sp + sdcp;
y := - sh * cd;
rsq := x *x + y * y;

IF rsq <> 0.0 THEN
	A := F_atan2(y,x);
ELSE
	A := 0.0;
END_IF


// The above formula assumes 0deg North and 90deg East. This
// must be corrected for VLT conventions 0deg is South. The 
// complete range of azimuth will be between 0-360.
// if (A < 0.0) A += vlt2PI;
A := - (A + GCL.C_PI);
IF A < 0.0 THEN
	A := A + GCL.C_2PI;
END_IF
A := F_vltMOD(A,GCL.C_2PI);

track.az_r 		:= A;
track.az_deg	:= track.az_r * GCL.C_RAD2DEG;

//
// CALC. Field Rotation 
//
track.fr_r		:= track.pa_r -  track.alt_r;
track.fr_deg	:= track.fr_r * GCL.C_RAD2DEG;

//////////////////////////
// Populate OUT structure
//////////////////////////

out_CcsDeterministic.current_observed_altaz[0]	:= track.alt_r;
out_CcsDeterministic.current_observed_altaz[1]	:= track.az_r;

out_CcsDeterministic.target_observed_altaz[0]	:= track.alt_r;
out_CcsDeterministic.target_observed_altaz[1]	:= track.az_r;

out_CcsDeterministic.time_tai	:= in_TimeStat.lrTaiUnixTimeinSecs;
out_CcsDeterministic.time_utc	:= in_TimeStat.lrTaiUnixTimeinSecs + time_data.leap_second;

out_CcsDeterministic.radec_at_altaz_at_requested_xy[0]	:= track.ra_r;
out_CcsDeterministic.radec_at_altaz_at_requested_xy[1]	:= track.dec_r;

out_CcsDeterministic.observed_altaz_at_requested_xy[0]	:= 0.0;
out_CcsDeterministic.observed_altaz_at_requested_xy[1]	:= 0.0;

out_CcsDeterministic.time_lst := track.ha_r + track.ra_r;

out_CcsDeterministic.parallactic_angle	:= track.pa_r;
out_CcsDeterministic.north_angle	:= track.pa_r + track.alt_r;
out_CcsDeterministic.pupil_angle	:= track.alt_r;



UserPointingKernel.parallactic_angle 	:= track.pa_r * GCL.C_RAD2DEG;
UserPointingKernel.north_angle 			:= out_CcsDeterministic.north_angle * GCL.C_RAD2DEG;
UserPointingKernel.pupil_angle 			:= track.alt_r * GCL.C_RAD2DEG;
UserPointingKernel.radec_at_altaz_at_requested_xy[0]:= F_astroRad2Hms(track.ra_r);
UserPointingKernel.radec_at_altaz_at_requested_xy[1]:= F_astroRad2Dms(track.dec_r);
UserPointingKernel.target_observed_altaz[0]		:= track.alt_r  * GCL.C_RAD2DEG;
UserPointingKernel.target_observed_altaz[1]		:= track.az_r  * GCL.C_RAD2DEG;
UserPointingKernel.current_observed_altaz[0]	:= track.alt_r  * GCL.C_RAD2DEG;
UserPointingKernel.current_observed_altaz[1]	:= track.az_r  * GCL.C_RAD2DEG;

M_TrkUpdate := TRUE;  // OK
END_METHOD

END_FUNCTION_BLOCK

// POUs/Functions/F_astroDms2rad
(*
 *   astroDms2rad   :   Convert an angle,given in user format, to radians.
 *   ===========
 *
 *   Given    :  angle      an angle as ddmmss.ttt (DegreesMinutesSecs)
 *   Returned :  rad        the angle as radians
 *
 *    The given angle, a floating value in the format DDMMSS.TTT, is 
 *    converted to radians. See also tcsSplitHms.
 *)
FUNCTION F_astroDms2rad : LREAL
VAR_INPUT
	angle:	LREAL;
END_VAR
VAR
	hh,hm,hs:	LREAL;
	ded,der:	LREAL;
END_VAR

(*
double astroDms2rad (double angle)
{
   double hh,hm,hs;
   double ded,der;
   double de2ra = 0.017453292519943;

   astroSplitHms(fabs_(angle),&hh,&hm,&hs);
   ded=hh + hm/60.0 + hs/3600.0;
   if (angle<0.0) ded=-ded; 
   der=ded*de2ra;
   
   return(der);
}*)

F_astroSplitHms(ABS(angle),h=>hh,m=>hm,sec=>hs);

ded	:= hh + hm/60.0 + hs/3600.0;

IF angle<0.0 THEN
	ded := -ded;
END_IF

der	:= ded * GCL.C_DEG2RAD;


F_astroDms2rad	:= der;

END_FUNCTION

// POUs/Functions/F_astroSplitHms
(*
 *   tcsSplitHms   :   Split an angle,given in user format, to its
 *   ===========      parts.
 *
 *   Given    :  angle      an angle as hhmmss.ttt (or ddmmss.tt)
 *   Returned :  h          hours (degrees)
 *               m          minutes (arcminutes)
 *               s          seconds (arcseconds)
 *
 *    The given time/angle, a floating value in the format HHMMSS.TTT, is split
 *    up in the parts HH, MM and SS.TTT (or DDMMSS.TTT if the input parameter
 *    is an angle).  
 *          NOTE:   if the given value is negative, all returned values 
 *    will also be negative! Which is may be not what you want, so take care of
 *    the sign outside of this function!
 * 
 *
 *   EXAMPLES
 *    Example 1:
 *     double time,h,m,s;
 *     time=123456.7;
 *     i=astroSplitHms(time,&h,&m,&s);
 *
 *        will return  h=12.0
 *                     m=34.0
 *                     s=56.7 
 *
 *
 *   Example 2:
 *     double time,h,m,s;
 *     time=345.0;
 *     i=astroSpltHms(time,&h,&m,&s);
 *
 *        will return  h=0.0
 *                     m=3.0
 *                     s=45.0 
 *
 *)
FUNCTION F_astroSplitHms : bool
VAR_INPUT
	angle:	LREAL;	// an angle as hhmmss.ttt (or ddmmss.tt)
END_VAR
VAR_OUTPUT
	h, m, sec:	LREAL;
END_VAR
VAR
   val:	LREAL;
   hours,minutes,seconds,t1,t2,t3:	LREAL;
 END_VAR

(*
void astroSplitHms (double angle, double *h, double *m, double *s)
{
   double val;
   double hour,min,sec,t1,t2,t3;
   
   val  = angle;  
   sec  = val - (int)(val/100.0)*100.0;    
   t1   = val-sec;
   t2   = t1 - (int)(t1/10000.0)*10000.0;
   min  = t2/100.0;
   t3   = val-sec-t2;
   hour = t3/10000;
   *h   = hour;
   *m   = min;
   *s   = sec;   
   return;
}
*)

val		:= angle;  
seconds	:= val - TRUNC_INT(val/100.0) * 100.0;    
t1		:= val - seconds;
t2		:= t1 - TRUNC_INT(t1/10000.0) * 10000.0;
minutes	:= t2/100.0;
t3		:= val - seconds - t2;
hours	:= t3/10000;

h	:= hours;
m	:= minutes;
sec	:= seconds;   

F_astroSplitHms	:= TRUE;

END_FUNCTION

// POUs/Functions/F_astroHms2rad
(*
 *   astroHms2rad   :   Convert a time/angle,given in user format, to radians.
 *   ===========
 *
 *   Given    :  angle      an angle as hhmmss.ttt (HoursMinutesSecs)
 *   Returned :  rad        the angle as radians
 *
 *    The given time/angle, a floating value in the format HHMMSS.TTT, is 
 *    converted to radians. See also tcsSplitHms
 *)
FUNCTION F_astroHms2rad : LREAL
VAR_INPUT
	angle:	LREAL;
END_VAR
VAR
	hh,hm,hs:	LREAL;
	rad,rar:	LREAL;
END_VAR

(*
double astroHms2rad (double angle)
{
   double hh,hm,hs;
   double rad,rar;
   double de2ra = 0.017453292519943;

   astroSplitHms(fabs_(angle),&hh,&hm,&hs);
   rad=(hh + hm/60.0 + hs/3600.0)*15.0;
   rar=rad*de2ra;
   if (angle<0.0) rar=-rar;
   
   return(rar);
}

*)

F_astroSplitHms(ABS(angle),h=>hh,m=>hm,sec=>hs);

rad	:= (hh + hm/60.0 + hs/3600.0) * 15.0;	// * 15.0 : 24h * 15 = 360 deg
rar	:= rad * GCL.C_DEG2RAD;

IF angle<0.0 THEN
	rar := -rar;
END_IF

F_astroHms2rad	:= rar;

END_FUNCTION

// POUs/Functions/F_astroRad2Hms
FUNCTION F_astroRad2Hms : LREAL
VAR_INPUT
	hh:	LREAL;	// angle in radians
END_VAR
VAR
	value:		LREAL;
	hours:		INT;
	minutes:	INT;
	seconds:	LREAL;
	
	sign:	int := 1;
END_VAR

IF hh < 0.0 THEN
	sign	:= -1;
	hh		:= -hh;
END_IF

value := hh / GCL.C_2PI * 24.0; 	// rad to hours


hours	:= TRUNC_INT(value);
minutes := TRUNC_INT((value - hours)*60.0);
seconds := (value - hours - minutes/60.0)*3600.0;

hours	:= hours * sign;	// put back the sign

					
F_astroRad2Hms	:= hours * 10000 + minutes * 100 + seconds;

END_FUNCTION

// POUs/Functions/F_astroRad2Dms
FUNCTION F_astroRad2Dms : LREAL
VAR_INPUT
	dd:	LREAL;	// angle in radians
END_VAR
VAR
	value:		LREAL;
	degrees:	INT;
	minutes:	INT;
	seconds:	LREAL;
	
	sign:	int := 1;
END_VAR

IF dd < 0.0 THEN
	sign	:= -1;
	dd		:= -dd;
END_IF

value := dd / GCL.C_2PI * 360.0; 	// rad to degrees


degrees	:= TRUNC_INT(value);
minutes := TRUNC_INT((value - degrees)*60.0);
seconds := (value - degrees - minutes/60.0)*3600.0;

					
F_astroRad2Dms	:= (degrees * 10000 + minutes * 100 + seconds) * sign;

END_FUNCTION

// POUs/Functions/F_timeUTCToMJD
(*
/*
 *****************************************************************************
 * timeUTCToMJD: convert struct ccsTIMEVAL into modified Julian date
 *
 *  IN   ut: time in UT
 *  OUT    : Modified julian date 
 ***************************************************************************** 
 */
*)
FUNCTION F_timeUTCToMJD : LREAL
VAR_INPUT
	ut:	T_TIMEVAL;
END_VAR
VAR
	mjd:	LREAL;
END_VAR

(*
DOUBLE timeUTCToMJD(vltTIMEVAL *ut)   /* time in UT                       */
    {
    DOUBLE mjd;                       /* modified julian date             */
   /*
    *# Get Julian Date from UT 
    */
    mjd = timeUTCToJD(ut);
    
   /*
    *# Convert Julian Date into Modified Julian Date according to the formula:
    *# MJD = JD - 2400000.5;
    */
    mjd-= CONST3;
    return(mjd);    
    }
*)

// Get Julian Date from UT 
mjd := F_timeUTCToJD(ut);

(*
*# Convert Julian Date into Modified Julian Date according to the formula:
*# MJD = JD - 2400000.5;
*)
F_timeUTCToMJD	:= mjd - GCL.C_CONST3;

END_FUNCTION

// POUs/Functions/F_timeUTCToJD
(*
/*
 *****************************************************************************
 * timeUTCToJD: convert struct ccsTIMEVAL into Julian date
 *
 *  IN   ut: time in UT
 *  OUT    : Julian date  
 ***************************************************************************** 
 */
*)
FUNCTION F_timeUTCToJD : LREAL
VAR_INPUT
	ut:	T_TIMEVAL;
END_VAR
VAR
	temp1:	LREAL;
END_VAR

(*
DOUBLE timeUTCToJD(vltTIMEVAL *ut)    /* time in UT                       */
    {
    DOUBLE jd;
    
   /*
    * CONST4 = jd(70-01-01 00:00:00.000000)
    */
    jd = CONST4 + (ut->tv_sec + ut->tv_usec/1000000.)/86400.;
    return(jd);
    }
*)

//F_timeUTCToJD := GCL.C_CONST4 + (UDINT_TO_REAL(ut.tv_sec) + DINT_TO_REAL(ut.tv_usec)/1000000.0)/86400.0;

temp1	:= DINT_TO_LREAL(ut.tv_usec)/1000000.0;
temp1	:= temp1 + UDINT_TO_LREAL(ut.tv_sec);

F_timeUTCToJD := GCL.C_CONST4 + (temp1)/86400.0;

END_FUNCTION

// POUs/Functions/F_timeGetUTC
(*
 *****************************************************************************
 * timeGetUTC: Get UTC time from TwinCAT DC time
 *
 *  IN   dcTime: TwinCAT DC time
 *  OUT  vltUTC: UTC time 
 ***************************************************************************** 
 *)
FUNCTION F_timeGetUTC : T_TIMEVAL
VAR_INPUT
	dcTime:   ULINT;
END_VAR
VAR
	ut:	T_TIMEVAL;
END_VAR

(*
HRESULT timeGetUTC(LONGLONG dcTime, vltTIMEVAL *vltUTC)
{
	HRESULT hr = S_OK; 
	
	// DC time is in nano seconds
	vltUTC->tv_sec = (LONGLONG)(dcTime/1000000000);
	vltUTC->tv_usec = (dcTime - (vltUTC->tv_sec * 1000000000))/1000;
	
	// Added offset between year 1970 and 2000 needed by the different references
	// used in UNIX and TWINCAT
	vltUTC->tv_sec += OFFSET_UNIX;
	return hr; 
}
*)

// DC time is in nano seconds
ut.tv_sec := ULINT_TO_UDINT(dcTime/1000000000);
ut.tv_usec := ULINT_TO_DINT((dcTime - UDINT_TO_ULINT(ut.tv_sec) * 1000000000)/1000);

// Added offset between year 1970 and 2000 needed by the different references
// used in UNIX and TWINCAT
ut.tv_sec := (ut.tv_sec + DINT_TO_UDINT(GCL.C_OFFSET_UNIX));

F_timeGetUTC	:= ut;

END_FUNCTION

// POUs/Functions/F_vltMod
FUNCTION F_vltMod : LREAL
VAR_INPUT
	number:		LREAL;
	divisor:	LREAL;
END_VAR
VAR
END_VAR

(*
static double vltMod(double number, double divisor)
{
    if (divisor == 0.0)
	return 0.0;
    return number - divisor * (int) (number / divisor);
}


*)

IF divisor = 0.0 THEN
	F_vltMod	:= 0.0;
ELSE
	F_vltMod	:= number - divisor * TRUNC_INT(number / divisor);
END_IF

END_FUNCTION

// POUs/Functions/F_slaPa
(*
/*+
**  - - - - - -
**   s l a P a
**  - - - - - -
**
**  HA, Dec to Parallactic Angle.
**
**  (double precision)
**
**  Given:
**     ha     d     hour angle in radians (geocentric apparent)
**     dec    d     declination in radians (geocentric apparent)
**     phi    d     observatory latitude in radians (geodetic)
**
**  The result is in the range -pi to +pi
**
*)
FUNCTION F_slaPa : LREAL
VAR_INPUT
	ha, dec, phi:	LREAL;
END_VAR
VAR
	cp, cqsz, sqsz:	LREAL;
	result:			LREAL;
END_VAR

(*
{
   double cp, cqsz, sqsz;

   cp = cos ( phi );
   sqsz = cp * sin ( ha );
   cqsz = sin ( phi ) * cos ( dec) - cp * sin ( dec) * cos ( ha );
   return ( ( sqsz != 0.0 || cqsz != 0.0 ) ? atan2 ( sqsz, cqsz ) : 0.0 );
}
*)

cp := COS ( phi );
sqsz := cp * SIN ( ha );
cqsz := SIN ( phi ) * COS ( dec) - cp * SIN ( dec) * COS ( ha );

//   return ( ( sqsz != 0.0 || cqsz != 0.0 ) ? atan2 ( sqsz, cqsz ) : 0.0 );
IF sqsz <> 0.0 OR cqsz <> 0.0 THEN
	result	:= F_atan2(sqsz, cqsz);
ELSE
	result	:= 0.0;
END_IF
	
F_slaPa	:= result;

END_FUNCTION

// POUs/Functions/F_atan2
// atan2(y,x)
FUNCTION F_atan2 : LREAL
VAR_INPUT
	y:	LREAL;
	x:	LREAL;
END_VAR
VAR
	atan2val:	LREAL;
END_VAR

IF (x > 0) THEN
	atan2val := ATAN(y/x);
ELSIF ((x < 0) AND (y >= 0)) THEN
	atan2val := ATAN(y/x) + GCL.C_PI;
ELSIF ((x < 0) AND (y < 0)) THEN
	atan2val := ATAN(y/x) - GCL.C_PI;
ELSIF ((x = 0) AND (y > 0)) THEN
	atan2val := GCL.C_PI2;
ELSIF ((x = 0) AND (y < 0)) THEN
	atan2val := -GCL.C_PI2;
ELSIF ((x = 0) AND (y = 0)) THEN
	atan2val := 1000;  //represents undefined
END_IF             

F_atan2	:= atan2val;

END_FUNCTION

// POUs/Functions/F_vltSign
FUNCTION F_vltSign : LREAL
VAR_INPUT
	number:	LREAL;
END_VAR
VAR
END_VAR

(*
static double vltSign(double number)
{
    if (number >= 0)
	return 1.0;
    return -1.0;
}
*)

IF number >= 0 THEN
	F_vltSign	:= 1.0;
ELSE
	F_vltSign	:= -1.0;
END_IF

END_FUNCTION

// POUs/Functions/F_DCTIME64_TO_ULINT
FUNCTION F_DCTIME64_TO_ULINT : ULINT
VAR_INPUT
	in:		T_DCTIME64;
END_VAR
VAR
	out:	ULINT;
END_VAR

memcpy (ADR(out), ADR(in), SIZEOF(in));
F_DCTIME64_TO_ULINT	:= out;

END_FUNCTION

// POUs/Functions/F_MOD
FUNCTION F_MOD : LREAL
VAR_INPUT
	A:	LREAL;
	B:	LREAL;
END_VAR
VAR
END_VAR

(*
#define vltMOD(A,B) 
((B)!=0.0?
	((A)*(B)>0.0?
		(A)-(B)*floor((A)/(B))
	else
		:(A)+(B)*floor(-(A)/(B)))
else
	:(A))
*)
IF B = 0.0 THEN
	F_MOD	:= A;
ELSE
	IF A * B >= 0.0 THEN
		F_MOD	:= A - B * TRUNC_INT(A / B);
	ELSE
		F_MOD	:= A + B * TRUNC_INT(-A / B);
	END_IF
END_IF

END_FUNCTION

// POUs/Functions/F_RAD2DMS_STRING
FUNCTION F_RAD2DMS_STRING : STRING
VAR_INPUT
	dec:	LREAL;
END_VAR
VAR
	value:		LREAL;
	degrees:	INT;
	minutes:	INT;
	seconds:	LREAL;
	
	sign:	int := 1;
	result:	STRING := '';
	
	fbFormat   : FB_FormatString;
END_VAR

IF dec < 0.0 THEN
	sign	:= -1;
	dec		:= -dec;
END_IF

value := dec * GCL.C_RAD2DEG; 	// rad to hours


degrees	:= TRUNC_INT(value);
minutes := TRUNC_INT((value - degrees)*60.0);
seconds := (value - degrees - minutes/60.0)*3600.0;

// We the calculation so far the value of 14.999999999 will result
// in 14:59:60.
// We want to correct it to 15:00:00.
IF seconds > 59.999 THEN
	seconds	:= 0.0;
	minutes	:= minutes + 1;
	IF minutes = 60 THEN
		minutes	:= 0;
		degrees	:= degrees + 1;
	END_IF
// Seconds should never be < 0.0. However, it happens due to rounding
// and the value could be ~ -1.0 e-12.
// Set it to zero in that case.
ELSIF seconds < 0.0 THEN
	seconds := 0.0;
END_IF

degrees	:= degrees * sign;	// put back the sign

// format a string like "+07:01:02.123"
fbFormat( sFormat  := '%+.3d:%.2d:%06.3f', 
					arg1 := F_INT(degrees), 
					arg2 := F_INT(minutes), 
					arg3 := F_LREAL(seconds),
					sOut => result);
					
F_RAD2DMS_STRING	:= result;

END_FUNCTION

// POUs/Functions/F_RAD2HMS_STRING
FUNCTION F_RAD2HMS_STRING : STRING
VAR_INPUT
	hh:	LREAL;
END_VAR
VAR
	value:		LREAL;
	hours:		INT;
	minutes:	INT;
	seconds:	LREAL;
	
	sign:	int := 1;
	result:	STRING := '';
	
	fbFormat   : FB_FormatString;
END_VAR

IF hh < 0.0 THEN
	sign	:= -1;
	hh		:= -hh;
END_IF

value := hh / GCL.C_2PI * 24.0; 	// rad to hours


hours	:= TRUNC_INT(value);
minutes := TRUNC_INT((value - hours)*60.0);
seconds := (value - hours - minutes/60.0)*3600.0;

// We the calculation so far the value of 14.999999999 will result
// in 14:59:60.
// We want to correct it to 15:00:00.
IF seconds > 59.999 THEN
	seconds	:= 0.0;
	minutes	:= minutes + 1;
	IF minutes = 60 THEN
		minutes	:= 0;
		hours	:= hours + 1;
	END_IF
// Seconds should never be < 0.0. However, it happens due to rounding
// and the value could be ~ -1.0 e-12.
// Set it to zero in that case.
ELSIF seconds < 0.0 THEN
	seconds := 0.0;
END_IF

hours	:= hours * sign;	// put back the sign

// format a string like "+07:01:02.123"
fbFormat( sFormat  := '%+.2d:%.2d:%06.3f', 
					arg1 := F_INT(hours), 
					arg2 := F_INT(minutes), 
					arg3 := F_LREAL(seconds),
					sOut => result);
					
F_RAD2HMS_STRING	:= result;

END_FUNCTION

// POUs/Functions/F_timeGetAbsoluteDcTime
(*
 *****************************************************************************
 * timeGetAbsoluteDcTime: Adjust DC time based on the external time signal
 *
 *  IN   ptptime    : External time signal
 *  IN   leapSecond : Leap Second 
 *  OUT  dcTIME     : Adjusted TwinCAT DC time
 ***************************************************************************** 
 *)
FUNCTION F_timeGetAbsoluteDcTime : BOOL
VAR_INPUT
	ptptime:			T_ASTRO_EL6688_DATA;
	nLeapSecond:		DINT;
	DcToExtTimeOffset:	LINT;
END_VAR
VAR_IN_OUT
	dcTime:   ULINT;
END_VAR
VAR
	val:		LINT	:= 0;
	diff:		LINT	:= 0;
	one_sec:	LINT	:= 1000000000;
END_VAR

(*
HRESULT timeGetAbsoluteDcTime(PTPTime ptptime, INT leapSecond, LONGLONG *dcTime)
{
	HRESULT hr = S_OK; 
	LONGLONG val = 0;
	LONGLONG diff = 0;
	LONGLONG ONE_SEC = 1000000000;
	
	// Check if external time signal is connected
	if (ptptime.not_connected)
		return S_FALSE;

	// If both variables are null means most probably they are not mapped.
	if (ptptime.internal == 0 || ptptime.external == 0)
		return S_FALSE;

	diff = (ptptime.internal - ptptime.external) + (ONE_SEC * leapSecond) + ptptime.dcTcOffset;
	*dcTime -=  diff;
	return hr;
}*)

// Check if external time signal is connected
IF ptptime.External_device_not_connected THEN
	F_timeGetAbsoluteDcTime := FALSE;
END_IF

// If both variables are null means most probably they are not mapped.
// TODO: Is it OR or AND ?
IF ptptime.Internal_time_stamp = 0  OR  ptptime.External_time_stamp = 0 THEN
	F_timeGetAbsoluteDcTime := FALSE;
END_IF

diff := (ULINT_TO_LINT(ptptime.Internal_time_stamp) - ULINT_TO_LINT(ptptime.External_time_stamp)) + 
		(one_sec * nLeapSecond) + DcToExtTimeOffset;

dcTime	:= dcTime - LINT_TO_ULINT(diff);

F_timeGetAbsoluteDcTime := TRUE;

END_FUNCTION

// POUs/Functions/F_timeGetDcTime
(*
 *****************************************************************************
 * timeGetDcTime: Get TwinCAT DC time from UTC time
 *
 *  IN   vltUTC: UTC time 
 *  OUT  dcTIME: TwinCAT DC time
 ***************************************************************************** 
 *)
FUNCTION F_timeGetDcTime : ULINT
VAR_INPUT
	ut:	T_TIMEVAL;
END_VAR
VAR
	val:   	ULINT := 0;
END_VAR

(*
HRESULT timeGetDcTime(vltTIMEVAL vltUTC, LONGLONG *dcTime)
{
	HRESULT hr = S_OK; 
	LONGLONG val = 0;
	val = vltUTC.tv_sec * 1000000000;
	val -= OFFSET_UNIX;
	*dcTime = val + vltUTC.tv_usec * 1000;
	return hr;
}
*)
val	:= ut.tv_sec * 1000000000;
val := val - DINT_TO_ULINT(GCL.C_OFFSET_UNIX);

F_timeGetDcTime	:= val + DINT_TO_ULINT(ut.tv_usec) * 1000;

END_FUNCTION

// POUs/Misc/FB_DIGITAL_SIGNAL_FILTER
// 
// Filtering of digital signal in order to remove glitches.
// It returns the dominant signal level (FALSE or TRUE) during
// the period of in_nPeriod_ms.
// It is a moving window. Therefore the output is 
// recalculated on every PLC cycle.
//
// Variable mapping:
//   i_bSig - Linked to the physical input signal coming from the switch.
//   q_bSig - Filtered output signal to be linked to motor switch var.
//
// Usage:
// 	df:	FB_DIGITAL_SIGNAL_FILTER;
//  df(in_nPeriod_ms:=nPeriod_ms);
//
FUNCTION_BLOCK FB_DIGITAL_SIGNAL_FILTER
VAR_INPUT
	// Sampling period [ms].
	// Resulting delay in signal change = MAX((period/2),in_nConseqToggle) + 1 cycle.
	// Switch detection error = (motor travel during (in_nPeriod_ms/2 + 1 cycle)).
	//
	// Example:
	//    PLC cycle = 1 ms
	//    in_nPeriod_ms = 7 ms  ==> nTotal = 7 (7 samples to process).
	//    in_nConseqToggle = 3 samples
	//    delay = MAX((7/2,3) + 1 = 3 + 1 = 4 PLC cycles
	//    The signal level that appeares >=3 times out of 5 samples,
	//    determines the resulting level TRUE/FALSE.
	//    Needed accuracy in switch detection = 0.6 um = 0.0006 mm.
	//    V = D / T  = 0.0006 / (4/1000) 
	//      = 0.0006 / (4/1000) = 0.0006 / 0.004 = 0.15 mm/sec
	//
	//    Conclusion: 
	//       The fine motor velocity for switch detection should be <= 0.15 mm/sec.
	//
	in_nPeriod_ms:		UINT := 5;	
	// Minimum consequtive toggles to toggle the filtered output.
	in_nConseqToggle:	UINT := 2;	
END_VAR
VAR
	//
	// Signals to map.
	//
	// Physical input signal that we want to process/filter.
	i_bSig     AT %I*: BOOL;
	// Generated filtered output signal.
	// The input signal, e.g., motor limit switch, should
	// be mapped to this signal instead of i_bSig.
	q_bSig     AT %Q*: BOOL;
	
	fbGetCurTaskIdx:	GETCURTASKINDEX;
	nCycleTime:			UDINT;	// Cycle time in microsec.

	nToggles: 		UINT := 0;
	nConseqToggles: UINT := 0;
	nTotal:			UINT;	// Total number of samples.
	// Number of consequtive same readings to swap the output.
	nToggleLimit: 	UINT := 1;	
	
	bReady:			BOOL;	// If TRUE, the FB is configured.
	
END_VAR

// Find out the total number of samples, i.e., PLC cycles.
IF NOT bReady	THEN

	// Get cycle time in microsec.
	// CycleTime in _TaskInfo is given in 100 ns. 1 us = 1000 ns
	fbGetCurTaskIdx();
	nCycleTime	:=  (TwinCAT_SystemInfoVarList._TaskInfo[fbGetCurTaskIdx.index].CycleTime)/10;

	// Get total number of samples to process
	nTotal	:= UDINT_TO_UINT(1000 * in_nPeriod_ms / nCycleTime);

	// There should be at least three samples
	nTotal	:= MAX(nTotal, 3);
	// Number of samples should be an odd number, i.e., 3, 5, 7, etc.
	IF nTotal MOD 2 = 0	THEN
		nTotal	:= nTotal + 1;
	END_IF

	// The number of consecutive cycles with opposite value
	// before swapping the output.
	nToggleLimit	:= nTotal / 2 + 1;

	bReady := TRUE;
	
	RETURN;
END_IF


//
// System is configured, i.e., ready to run.
//

//
// Check if the input signal is the same as the filtered output.
//
IF i_bSig <> q_bSig THEN
	IF nToggles > 1  AND  nConseqToggles = 0	THEN
		// The previous non-toggle lasted only one sample,
		// This was a glitch.
		// Discard it by incrementing toggles by 2 
		// {this one plus the previous one)
		nToggles 		:= nToggles + 2;
	ELSE
		nToggles 		:= nToggles + 1;
	END_IF
	
	// Increment the number of consequtive toggles.
	nConseqToggles	:= nConseqToggles + 1;
	// At least in_nConseqToggle consequtive toggle readings
	// needed to toggle the filtered signal.
	IF nToggles >= nToggleLimit  AND  nConseqToggles >= in_nConseqToggle 	THEN
		// Toggle output
		q_bSig 			:= NOT q_bSig;
		nToggles		:= 0;
		nConseqToggles	:= 0;	
	END_IF
ELSE
	IF nToggles = 1  AND  nConseqToggles = 1	THEN
		// There was a toggle in the previous sample,
		// but now there is no toggle.
		// This was a glitch.
		nToggles		:= 0;	
	ELSE
		// Decrement the number of toggles.
		IF nToggles > 1	THEN
			nToggles := nToggles - 1;
		ELSE	
			nToggles := 0;
		END_IF
	END_IF
	
	// Reset the counter for consequtive toggles.
	nConseqToggles	:= 0;	
END_IF

END_FUNCTION_BLOCK

// POUs/Motor/FB_MOTOR
FUNCTION_BLOCK FB_MOTOR EXTENDS FB_MOTOR_BASE
VAR_INPUT
	{attribute 'OPC.UA.DA' := '0'}
	sName:			STRING	:= 'Motor';	(* Default Motor name *)
	{attribute 'OPC.UA.DA' := '0'}
	nNOVRAM_DevId:	UDINT	:= 0;		(* NOVRAM device ID - normally 4 *)
	{attribute 'OPC.UA.DA' := '0'}
	nNOVRAM_Offset:	UDINT	:= 0;		(* NOVRAM offset where motor configuration is stored *)
END_VAR
VAR_OUTPUT
END_VAR
VAR
	
	(***** Local variables *****)
	{attribute 'OPC.UA.DA' := '0'}
	toutCmd:	TON;
	{attribute 'OPC.UA.DA' := '0'}
	trg:		R_TRIG;
	{attribute 'OPC.UA.DA' := '0'}
	timer:		TON;	(* Timer for measuring duration of events *)
	{attribute 'OPC.UA.DA' := '0'}
	nState_Init:			INT := MOTOR_INIT_STATE_RESET;		// State of ActivityInitializing
	{attribute 'OPC.UA.DA':='0'}
	nState_Reset:			INT := MOTOR_RESET_STATE_START;
	{attribute 'OPC.UA.DA':='0'}
	nState_PreInit:			INT	:= MOTOR_PRE_INIT_STATE_START;
	{attribute 'OPC.UA.DA':='0'}
	nState_InitSeq:			INT := MOTOR_INIT_SEQ_STATE_START;
	{attribute 'OPC.UA.DA':='0'}
	nState_PostInit:		INT	:= MOTOR_POST_INIT_STATE_START;
	{attribute 'OPC.UA.DA':='0'}
	nState_Moving:			INT := MOTOR_MOVING_STATE_WAIT_BRAKES;		// State of ActivityMoving
	{attribute 'OPC.UA.DA':='0'}
	nState_MovingNext:		INT := MOTOR_MOVING_STATE_WAIT_ABSOLUTE;	// Next state after checking brakes


	(***** Physical signals - to be mapped!!! *****)

	(* Outputs *)
	{attribute 'OPC.UA.DA' := '0'}
	q_bBrake_Ctrl	AT %Q*:	BOOL;				(* Brake control signal - DIGITAL OUT *)


	(* Inputs *)	
	{attribute 'OPC.UA.DA':='0'}
	switches		AT %I*:	T_MOTOR_SWITCHES;	(* Limit switches *)
	{attribute 'OPC.UA.DA':='0'}
	i_bInPos		AT %I*:	BOOL;				(* In-position signal - DIGITAL IN *)
	{attribute 'OPC.UA.DA':='0'}
	i_bBrake_Stat	AT %I*:	BOOL;				(* Brake feedback signal - DIGITAL IN *)
	{attribute 'OPC.UA.DA':='0'}
	i_nInfoData1	AT %I*:	UINT;				(* Info data 1 from Motor I/O terminal *)
	{attribute 'OPC.UA.DA':='0'}
	i_nInfoData2	AT %I*:	UINT;				(* Info data 2 from Motor I/O terminal *)
	{attribute 'OPC.UA.DA':='0'}
	i_nSoE_DriveStatus	AT %I*:	UINT;			(* Drive Status. SoE Drives, e.g. AX5000, ONLY!!! *)
	{attribute 'OPC.UA.DA':='0'}
	i_nSoE_PowerStatus	AT %I*:	INT;			(* Power Status. SoE Drives, e.g. AX5000, ONLY!!! *)

	{attribute 'OPC.UA.DA' := '0'}
	i_nCouplerState	AT %I*: 		UINT;	(* Link it to Coupler->InfoData->State *)

	{attribute 'OPC.UA.DA' := '0'}
	Axis:  		AXIS_REF;


(* Ctrl parameters used by ctrl.bExecute *)
	{attribute 'OPC.UA.DA':='0'}
	nCurDirection:	DINT	:=	INT_TO_DINT(MC_Positive_Direction);
	{attribute 'OPC.UA.DA':='0'}
	lrCurVelocity:	LREAL	:=	0.0;
	

(* Function block instances *)

	{attribute 'OPC.UA.DA' := '0'}
	fbHalt: 	           		MC_Halt;
	{attribute 'OPC.UA.DA' := '0'}
	fbSoEReset: 	           	FB_SoEReset;
	{attribute 'OPC.UA.DA' := '0'}
	fbResetError: 	           	MC_Reset;
	{attribute 'OPC.UA.DA' := '0'}
	fbMovePos_1:  	 			MC_MoveAbsolute;
	{attribute 'OPC.UA.DA' := '0'}
	fbMovePos_2:  	 			MC_MoveAbsolute;
	{attribute 'OPC.UA.DA' := '0'}
	ptr_fbMovePos: POINTER TO 	MC_MoveAbsolute := ADR(fbMovePos_1);
	{attribute 'OPC.UA.DA' := '0'}
	fbMoveVel_1:  	 			MC_MoveVelocity;
	{attribute 'OPC.UA.DA' := '0'}
	fbMoveVel_2:				MC_MoveVelocity;
	{attribute 'OPC.UA.DA' := '0'}
	ptr_fbMoveVel: POINTER TO 	MC_MoveVelocity := ADR(fbMoveVel_1);
	{attribute 'OPC.UA.DA' := '0'}
	fbMoveOpt_1:				MC_MoveModulo;
	{attribute 'OPC.UA.DA' := '0'}
	fbMoveOpt_2:				MC_MoveModulo;
	{attribute 'OPC.UA.DA' := '0'}
	ptr_fbMoveOpt: POINTER TO 	MC_MoveModulo := ADR(fbMoveOpt_1);
	{attribute 'OPC.UA.DA' := '0'}
	fbStop:						MC_Stop;
	{attribute 'OPC.UA.DA' := '0'}
	fbSetActualPosition:		MC_SetPosition;

	(* There are two FB's per Pos, Vel and circular-optimised. Keep track which one is active. *)
	{attribute 'OPC.UA.DA':='0'}
	nFbPos:		INT := 1; 
	{attribute 'OPC.UA.DA':='0'}
	nFbVel:		INT := 1; 
	{attribute 'OPC.UA.DA':='0'}
	nFbOpt:		INT := 1; 
	
	(* Temporary vars for finding shortest way for circular-optimised with backlash compensation *)
	{attribute 'OPC.UA.DA':='0'}
	nOptDir:		MC_Direction;	(* Optimised direction *)
	{attribute 'OPC.UA.DA':='0'}
	lrTmpDist1:		LREAL;
	{attribute 'OPC.UA.DA':='0'}
	lrTmpDist2:		LREAL;
	{attribute 'OPC.UA.DA':='0'}
	lrTmpPos1:		LREAL;
	{attribute 'OPC.UA.DA':='0'}
	lrTmpPos2:		LREAL;
	
	(* NOVRAM Handling *)
	{attribute 'OPC.UA.DA':='0'}
	bNOVRAM_Error:		BOOL := FALSE;	(* NOVRAM error active flag *)
	{attribute 'OPC.UA.DA':='0'}
	bNOVRAM_Loaded:		BOOL := FALSE;	(* Flag if NOVRAM has been loaded *)
	{attribute 'OPC.UA.DA':='0'}
	nNOVRAM_State_R:	UINT := 0;		(* NOVRAM Read state *)
	{attribute 'OPC.UA.DA':='0'}
	nNOVRAM_State_W:	UINT := 0;		(* NOVRAM Write state *)
	{attribute 'OPC.UA.DA':='0'}
	stMotorCfg_NOVRAM:	T_MOTOR_CFG;	(* NOVRAM copy of motor config. Read on First PLC cycle. *)

	{attribute 'OPC.UA.DA':='0'}
	fbNovReadWrite: 	Tc2_IoFunctions.FB_NovRamReadWriteEx;

END_VAR

// Basic configuration, executed once internally
M_Configure();

// Increment alive counter
stat.nCounter	:= stat.nCounter + 1;

(* Read motor status *)
Axis.ReadStatus();


(* Update states of Limit Switches *)
M_UpdateSwitches();

// 	Enable directions based on the state of STOP switches. 
//	Active LSTOP switch (stat.bStopSwitchNeg) disables motion in negative direction
//	Active USTOP switch (stat.bStopSwitchPos) disables motion in positive direction
Axis.PlcToNc.ControlDWord := AxisSetControllerEnable(Axis.PlcToNc.ControlDWord, stat.bEnabled);
Axis.PlcToNc.ControlDWord := AxisSetFeedEnableMinus(Axis.PlcToNc.ControlDWord, (NOT stat.bStopSwitchNeg));
Axis.PlcToNc.ControlDWord := AxisSetFeedEnablePlus(Axis.PlcToNc.ControlDWord,  (NOT stat.bStopSwitchPos));

(* 
	If both limit switches are active ((LSTOP & USTOP) or (LHW & UHW)), disable the motor and set error. 
	Do this check after NOVRAM configuration has been loaded. Doing it earlier
	could report some non-existing errors.
*)
IF	bNOVRAM_Loaded THEN
	IF 	stat.signals[E_MOTOR_SWITCH_INDEX.LSTOP].bActive AND stat.signals[E_MOTOR_SWITCH_INDEX.USTOP].bActive 	THEN
		stat.bEnabled 				:= FALSE;
		Axis.PlcToNc.ControlDWord 	:= AxisSetFeedEnableMinus(Axis.PlcToNc.ControlDWord, FALSE);
		Axis.PlcToNc.ControlDWord 	:= AxisSetFeedEnablePlus(Axis.PlcToNc.ControlDWord,  FALSE);
		M_SetError(E_MOTOR_ERROR.STOP_LIMITS_BOTH, 'ERROR: Both LSTOP and USTOP limits active. Motor disabled.');
	ELSIF 	stat.signals[E_MOTOR_SWITCH_INDEX.LHW].bActive AND stat.signals[E_MOTOR_SWITCH_INDEX.UHW].bActive 	THEN
		stat.bEnabled 				:= FALSE;
		Axis.PlcToNc.ControlDWord 	:= AxisSetFeedEnableMinus(Axis.PlcToNc.ControlDWord, FALSE);
		Axis.PlcToNc.ControlDWord 	:= AxisSetFeedEnablePlus(Axis.PlcToNc.ControlDWord,  FALSE);
		M_SetError(E_MOTOR_ERROR.HW_LIMITS_BOTH, 'ERROR: Both LHW and UHW limits active. Motor disabled.');
	END_IF
END_IF

(* Set velocity override to 100% *)
Axis.PlcToNc.Override := 1000000;


(* Check that Axis is in READY State *)
stat.bAxisReady := AxisIsReady(Axis.NcToPlc.StateDWord);

(* Read actual position and velocity. Circular optimised has normalised value *)
stat.lrPosActual	:= M_GetActualPos();
stat.lrVelActual	:= Axis.NcToPlc.ActVelo;
stat.lrPosError		:= Axis.NcToPlc.PosDiff;

(* Read Info data parameters *)
stat.nInfoData1	:= UINT_TO_INT(i_nInfoData1);
stat.nInfoData2	:= UINT_TO_INT(i_nInfoData2);

(* If brakes are not used, release them. Brakes are hard-coded to active low! *)
(*
This seems to not be needed since q_bBrake_Ctrl should not be mapped!
IF NOT cfg.bUseBrake THEN
	q_bBrake_Ctrl	:= M_GetLogicalState(state:= FALSE, activeLow:= TRUE);
END_IF
*)

(* Get the state of the brake *)
stat.bBrakeActive	:= M_GetLogicalState(state:= i_bBrake_Stat, activeLow:= cfg.bActiveLowBrake);

// Get the In-Position status
stat.bInPosition	:= M_GetLogicalState(i_bInPos, cfg.bActiveLowInPos);

(* === Check for commands and internal events to be processed === *)
CheckForEvents();

(* === Process events according to the State Machine === *)
ProcessEvents();

METHOD ActionClearNOVRAM
VAR_INPUT
END_VAR
SetAction('ActionClearNOVRAM');

// Log event
M_LogEventStart('CLEAR NOVRAM');

M_NOVRAM_Clear(FALSE);		// Trigger M_NOVRAM_Clear()
END_METHOD

METHOD ActionErrExecute
VAR
END_VAR
SetAction('ActionErrExecute');

IF nEvent = E_MOTOR_EVENT.TIMEOUT_MOVE THEN
	M_SetStatus(E_MOTOR_ERROR.TIMEOUT_MOVE);
ELSIF nEvent = E_MOTOR_EVENT.TIMEOUT_SETPOS THEN
	M_SetStatus(E_MOTOR_ERROR.TIMEOUT_SETPOS);
END_IF
END_METHOD

METHOD ActionInitAbort
VAR_INPUT
END_VAR
SetAction('ActionInitAbort');

M_LogEventGeneral('Aborting INIT...');

// Set Error Status
M_SetStatus(E_MOTOR_ERROR.INIT_ABORTED);

// Apply brakes. Brakes are hard-coded to active low!
q_bBrake_Ctrl	:= M_GetLogicalState(state:= TRUE, activeLow:= TRUE);


// Reset the timer for the command
toutCmd(IN:=FALSE);
toutCmd(IN:=TRUE,PT:=UDINT_TO_TIME(cfg.nTimeoutInit));

// Restart HALT FB
fbHalt(Execute:=FALSE, Axis:=Axis);
//fbHalt(Execute:=TRUE, Axis:=Axis);

(*
IF NOT Axis.Status.NotMoving THEN
	// Restart the timer
	toutCmd(IN:=TRUE,PT:=DINT_TO_TIME(cfg.nTimeoutInit));
END_IF
*)

stat.bInitialised	:= FALSE;
//stat.bEnabled		:= FALSE;
stat.nInitStep		:= 0;
END_METHOD

METHOD ActionInitComplete
VAR_INPUT
END_VAR
SetAction('ActionInitComplete');

// Log event
M_LogEventEnd('INIT');

(* reply OK *)
stat.nErrorCode		:= E_MOTOR_ERROR.OK;
stat.sErrorText		:= 'OK';

(* Reset the timer action *)
toutCmd(IN:=FALSE);
END_METHOD

METHOD ActionInitExecute
VAR_INPUT
END_VAR
SetAction('ActionInitExecute');

// Log event
M_LogEventStart('INIT');

// Set starting states for all methods to be executed in INIT
nState_Init		:= MOTOR_INIT_STATE_RESET;
nState_Reset	:= MOTOR_RESET_STATE_START;
nState_InitSeq	:= MOTOR_INIT_SEQ_STATE_START;
nState_PreInit	:= MOTOR_PRE_INIT_STATE_START;
nState_PostInit	:= MOTOR_POST_INIT_STATE_START;

stat.bInitialised	:= FALSE;	// Clear the initialised flag

// Enable motor
stat.bEnabled	:= TRUE;

// Release brakes. Brakes are hard-coded to active low!
q_bBrake_Ctrl	:= M_GetLogicalState(state:= FALSE, activeLow:= TRUE);

// Start the cmd timer.
// Give 5 sec more than the timeout for INIT sequence
toutCmd(IN:=FALSE);
toutCmd(IN:=TRUE,PT:=UDINT_TO_TIME(cfg.nTimeoutInit+5000));
END_METHOD

METHOD ActionInitReject
VAR_INPUT
END_VAR
SetAction('ActionInitReject');

(* Reject an INIT command since another one is in progress. *)
(* do not reset the timer ... *)
END_METHOD

METHOD ActionMoveExecute
VAR_INPUT
END_VAR
SetAction('ActionMoveExecute');

(* Clear the error *)
M_SetStatus(E_MOTOR_ERROR.OK);

(* 
	MOVE RELATIVE is converted to MOVE ABSOLUTE
	We just add the offset to the current position and move absolute!
*)
IF ctrl.nMoveType = E_MOTOR_MOVE_TYPE.RELATIVE THEN
	M_LogEventMoveRel(ctrl.lrOffset, stat.lrPosActual, ctrl.lrVelocity);
	M_LogEventDebug('MOVEREL converted to MOVEABS');
	ctrl.lrPosition		:= stat.lrPosActual + ctrl.lrOffset;	(* Set new absolute position *)
	ctrl.nMoveType 		:= E_MOTOR_MOVE_TYPE.ABSOLUTE; 
END_IF


// Handling of Locked function. 
// If the motor is locked, there is no need to prepare anything here.
// We just exit this method.
// Method ActivityMoving() will do a check and set error, if needed.
IF 	cfg.bLock THEN
	// Nothing to do - exit this method.
	RETURN;
END_IF


// Variable nState_MovingNext is used to set the type of wait for the end of motion.
// It can be either 
//	- MOTOR_MOVING_STATE_WAIT_ABSOLUTE, 
//	- MOTOR_MOVING_STATE_WAIT_OPTIMISED or 
//	- MOTOR_MOVING_STATE_WAIT_VELOCITY.
// However, prior to moving, we handle ENABLE, Brakes and USER_PRE_MOVE
// Variable nState_Moving is used for that purpose.


IF 	(ctrl.nMoveType = E_MOTOR_MOVE_TYPE.ABSOLUTE OR ctrl.nMoveType = E_MOTOR_MOVE_TYPE.TRACKING) AND  
	cfg.nAxisType <> E_MOTOR_AXIS_TYPE.CIRCULAR_OPTIMISED  THEN
	stat.nMode 		:= E_MOTOR_MODE.POS;
	stat.nErrorCode := 0;
	// If brakes are used, this will be the next step in ActivityMoving() after brake release.
	nState_MovingNext := MOTOR_MOVING_STATE_WAIT_ABSOLUTE; 
	
	(*
		Motor move has two steps in case of backlash compensation.
		If there is no compensation, we start from the second (end)  step.
		
	 	Check if we need a two step movement.
		Adjust the target position to a multiple of the scaling factor, 
		i.e. whole number of encoder or motor steps.
	*)
	IF 	(cfg.lrBacklash > 0.0 AND (stat.lrPosActual - ctrl.lrPosition < cfg.lrBacklash)) OR
		(cfg.lrBacklash < 0.0 AND (stat.lrPosActual - ctrl.lrPosition > cfg.lrBacklash)) THEN
		stat.nBacklashStep	:= 1;
		stat.lrPosTarget 	:= LREAL_TO_DINT((ctrl.lrPosition + cfg.lrBacklash) / stat.axis.lrScaleFactor) * stat.axis.lrScaleFactor;
	ELSE
		stat.nBacklashStep 	:= 2;
		stat.lrPosTarget 	:= LREAL_TO_DINT(ctrl.lrPosition / stat.axis.lrScaleFactor) * stat.axis.lrScaleFactor;
	END_IF


	(* 	
		Find currently running FB and swap to the other one.
		This way we can update position and velocity on the fly.
		Execute the corresponding MC_MoveAbsolute with the flag Execute = FALSE.
		Next call with Execute = TRUE will trigger execution of the FB. 
	*)
	IF nFbPos = 1 THEN
		nFbPos 			:= 2;
		ptr_fbMovePos	:= ADR(fbMovePos_2);
	ELSE
		nFbPos 			:= 1;
		ptr_fbMovePos	:= ADR(fbMovePos_1);
	END_IF

	// Triger motor move by toggling the Execute flag
	ptr_fbMovePos^(
		Execute			:= FALSE,
		Axis			:= Axis,
		Position		:= stat.lrPosTarget,
		Velocity		:= ctrl.lrVelocity,
		Acceleration 	:= stat.axis.lrAccel,
		Deceleration 	:= stat.axis.lrDecel,
		Jerk			:= stat.axis.lrJerk,
		BufferMode		:= MC_Aborting);

	(* The motor is moving in Position mode *)
	M_LogEventMoveAbs(ctrl.lrPosition, ctrl.lrVelocity);
	M_SetStatusDescription(E_MOTOR_STATUS.MOVING, 'Moving in Position');

	(* ============= MOVE ABSOLUTE - OPTIMISED =============== *)
ELSIF 	(ctrl.nMoveType = E_MOTOR_MOVE_TYPE.ABSOLUTE OR ctrl.nMoveType = E_MOTOR_MOVE_TYPE.TRACKING)  AND  
		cfg.nAxisType  = E_MOTOR_AXIS_TYPE.CIRCULAR_OPTIMISED  THEN
	stat.nMode 		:= E_MOTOR_MODE.POS;
	stat.nErrorCode := 0;
	// If brakes are used, this will be the next step in ActivityMoving() after brake release.
	nState_MovingNext := MOTOR_MOVING_STATE_WAIT_OPTIMISED; 
	
	// Normalise set position
	ctrl.lrPosition	:= M_GetOptimisedPosition(ctrl.lrPosition);

	(*
		Motor move has two steps in case of backlash compensation.
		If there is no compensation, we start from the second (end)  step.
	 
		Check if we need a two step movement. 
	*)
	IF 	cfg.lrBacklash <> 0.0 THEN
		(* 
			Get the two positions in the 2-step movement. Pos2 is the final position.
			Then we check if one step is enough.
		*)
		lrTmpPos1	:= M_GetOptimisedPosition(lrPos:=(ctrl.lrPosition + cfg.lrBacklash));
		lrTmpPos2	:= M_GetOptimisedPosition(lrPos:=(ctrl.lrPosition));
		// Adjust the target position to a multiple of the scaling factor, i.e. whole number of encoder or motor steps
		lrTmpPos2 	:= LREAL_TO_DINT(lrTmpPos2 / stat.axis.lrScaleFactor) * stat.axis.lrScaleFactor;
		(* Get the distance from the current to the first position, and from the current to the final position. *)
		lrTmpDist1	:= M_GetOptimisedDistance(lrPos1:=stat.lrPosActual, lrPos2:=lrTmpPos1);
		lrTmpDist2	:= M_GetOptimisedDistance(lrPos1:=stat.lrPosActual, lrPos2:=lrTmpPos2);

